LIN {X 0,Y 523.921,Z 257.848,A -85,B 0,C 180,E1 -4821.081,E2 -4821.081} C_VEL
LIN {X 0,Y 523.901,Z 257.849,A -85,B 0,C 180,E1 -4823.825,E2 -4823.825} C_VEL
LIN {X 0,Y 523.947,Z 257.848,A -85,B 0,C 180,E1 -4826.636,E2 -4826.636} C_VEL
LIN {X 0,Y 523.962,Z 257.841,A -85,B 0,C 180,E1 -4829.356,E2 -4829.356} C_VEL
LIN {X 0,Y 523.951,Z 257.849,A -85,B 0,C 180,E1 -4832.288,E2 -4832.288} C_VEL
LIN {X 0,Y 523.949,Z 257.848,A -85,B 0,C 180,E1 -4834.581,E2 -4834.581} C_VEL
LIN {X 0,Y 523.965,Z 257.93,A -85,B 0,C 180,E1 -4836.952,E2 -4836.952} C_VEL
LIN {X 0,Y 525.894,Z 266.836,A -85,B 0,C 180,E1 -4838.612,E2 -4838.612} C_VEL
LIN {X 0,Y 528.548,Z 277.959,A -85,B 0,C 180,E1 -4838.908,E2 -4838.908} C_VEL
LIN {X 0,Y 527.339,Z 416.797,A -85,B 0,C 180,E1 -4840.955,E2 -4840.955} C_VEL
LIN {X 0,Y 527.174,Z 435.165,A -85,B 0,C 180,E1 -4841.271,E2 -4841.271} C_VEL
LIN {X 0,Y 526.901,Z 450.096,A -85,B 0,C 180,E1 -4841.682,E2 -4841.682} C_VEL
LIN {X 0,Y 526.575,Z 464.31,A -85,B 0,C 180,E1 -4842.223,E2 -4842.223} C_VEL
LIN {X 0,Y 526.183,Z 478.273,A -85,B 0,C 180,E1 -4842.911,E2 -4842.911} C_VEL
LIN {X 0,Y 525.76,Z 492.557,A -85,B 0,C 180,E1 -4843.797,E2 -4843.797} C_VEL
LIN {X 0,Y 525.311,Z 505.414,A -85,B 0,C 180,E1 -4844.778,E2 -4844.778} C_VEL
LIN {X 0,Y 524.873,Z 517.153,A -85,B 0,C 180,E1 -4845.855,E2 -4845.855} C_VEL
LIN {X 0,Y 524.507,Z 527.829,A -85,B 0,C 180,E1 -4847.03,E2 -4847.03} C_VEL
LIN {X 0,Y 524.096,Z 538.235,A -85,B 0,C 180,E1 -4848.395,E2 -4848.395} C_VEL
LIN {X 0,Y 523.9,Z 546.784,A -85,B 0,C 180,E1 -4849.761,E2 -4849.761} C_VEL
LIN {X 0,Y 523.65,Z 553.936,A -85,B 0,C 180,E1 -4851.121,E2 -4851.121} C_VEL
LIN {X 0,Y 523.526,Z 560.464,A -85,B 0,C 180,E1 -4852.673,E2 -4852.673} C_VEL
LIN {X 0,Y 523.483,Z 565.622,A -85,B 0,C 180,E1 -4854.22,E2 -4854.22} C_VEL
LIN {X 0,Y 523.335,Z 568.597,A -85,B 0,C 180,E1 -4855.378,E2 -4855.378} C_VEL
LIN {X 0,Y 523.389,Z 571.449,A -85,B 0,C 180,E1 -4856.921,E2 -4856.921} C_VEL
LIN {X 0,Y 523.273,Z 573.167,A -85,B 0,C 180,E1 -4858.46,E2 -4858.46} C_VEL
LIN {X 0,Y 523.246,Z 573.806,A -85,B 0,C 180,E1 -4859.999,E2 -4859.999} C_VEL
LIN {X 0,Y 523.273,Z 573.231,A -85,B 0,C 180,E1 -4861.539,E2 -4861.539} C_VEL
LIN {X 0,Y 523.391,Z 571.557,A -85,B 0,C 180,E1 -4863.078,E2 -4863.078} C_VEL
LIN {X 0,Y 523.333,Z 568.774,A -85,B 0,C 180,E1 -4864.621,E2 -4864.621} C_VEL
LIN {X 0,Y 523.441,Z 564.656,A -85,B 0,C 180,E1 -4866.165,E2 -4866.165} C_VEL
LIN {X 0,Y 523.557,Z 559.289,A -85,B 0,C 180,E1 -4867.714,E2 -4867.714} C_VEL
LIN {X 0,Y 523.705,Z 552.375,A -85,B 0,C 180,E1 -4869.266,E2 -4869.266} C_VEL
LIN {X 0,Y 523.949,Z 544.953,A -85,B 0,C 180,E1 -4870.628,E2 -4870.628} C_VEL
LIN {X 0,Y 524.199,Z 536.232,A -85,B 0,C 180,E1 -4871.966,E2 -4871.966} C_VEL
LIN {X 0,Y 524.52,Z 526.84,A -85,B 0,C 180,E1 -4873.166,E2 -4873.166} C_VEL
LIN {X 0,Y 524.9,Z 516.03,A -85,B 0,C 180,E1 -4874.341,E2 -4874.341} C_VEL
LIN {X 0,Y 525.356,Z 503.897,A -85,B 0,C 180,E1 -4875.437,E2 -4875.437} C_VEL
LIN {X 0,Y 525.813,Z 491.098,A -85,B 0,C 180,E1 -4876.4,E2 -4876.4} C_VEL
LIN {X 0,Y 526.27,Z 478.382,A -85,B 0,C 180,E1 -4877.185,E2 -4877.185} C_VEL
LIN {X 0,Y 526.614,Z 464.639,A -85,B 0,C 180,E1 -4877.875,E2 -4877.875} C_VEL
LIN {X 0,Y 526.981,Z 448.493,A -85,B 0,C 180,E1 -4878.49,E2 -4878.49} C_VEL
LIN {X 0,Y 527.289,Z 433.513,A -85,B 0,C 180,E1 -4878.893,E2 -4878.893} C_VEL
LIN {X 0,Y 527.459,Z 412.098,A -85,B 0,C 180,E1 -4879.248,E2 -4879.248} C_VEL
LIN {X 0,Y 528.568,Z 278.087,A -85,B 0,C 180,E1 -4881.184,E2 -4881.184} C_VEL
LIN {X 0,Y 525.425,Z 265.012,A -85,B 0,C 180,E1 -4881.534,E2 -4881.534} C_VEL
LIN {X 0,Y 523.937,Z 257.848,A -85,B 0,C 180,E1 -4882.812,E2 -4882.812} C_VEL
LIN {X 0,Y 523.91,Z 257.851,A -85,B 0,C 180,E1 -4883.324,E2 -4883.324} C_VEL
LIN {X 0,Y 523.244,Z 257.937,A -85,B 0,C 180,E1 -4883.965,E2 -4883.965} C_VEL
LIN {X 0,Y 520.418,Z 258.288,A -85,B 0,C 180,E1 -4885.006,E2 -4885.006} C_VEL
LIN {X 0,Y 518.024,Z 258.585,A -85,B 0,C 180,E1 -4885.845,E2 -4885.845} C_VEL
LIN {X 0,Y 516.984,Z 258.71,A -85,B 0,C 180,E1 -4886.492,E2 -4886.492} C_VEL
LIN {X 0,Y 516.893,Z 258.72,A -85,B 0,C 180,E1 -4886.711,E2 -4886.711} C_VEL
LIN {X 0,Y 516.909,Z 258.721,A -85,B 0,C 180,E1 -4889.522,E2 -4889.522} C_VEL
LIN {X 0,Y 516.895,Z 258.719,A -85,B 0,C 180,E1 -4892.542,E2 -4892.542} C_VEL
LIN {X 0,Y 516.863,Z 258.724,A -85,B 0,C 180,E1 -4895.328,E2 -4895.328} C_VEL
LIN {X 0,Y 516.877,Z 258.728,A -85,B 0,C 180,E1 -4897.942,E2 -4897.942} C_VEL
LIN {X 0,Y 516.881,Z 258.72,A -85,B 0,C 180,E1 -4900.741,E2 -4900.741} C_VEL
LIN {X 0,Y 516.861,Z 258.722,A -85,B 0,C 180,E1 -4902.832,E2 -4902.832} C_VEL
LIN {X 0,Y 516.893,Z 258.718,A -85,B 0,C 180,E1 -4905.006,E2 -4905.006} C_VEL
LIN {X 0,Y 516.911,Z 258.718,A -85,B 0,C 180,E1 -4908.398,E2 -4908.398} C_VEL
LIN {X 0,Y 516.877,Z 258.723,A -85,B 0,C 180,E1 -4911.283,E2 -4911.283} C_VEL
LIN {X 0,Y 516.868,Z 258.724,A -85,B 0,C 180,E1 -4914.219,E2 -4914.219} C_VEL
LIN {X 0,Y 516.877,Z 258.721,A -85,B 0,C 180,E1 -4917.051,E2 -4917.051} C_VEL
LIN {X 0,Y 516.887,Z 258.727,A -85,B 0,C 180,E1 -4919.795,E2 -4919.795} C_VEL
LIN {X 0,Y 516.895,Z 258.719,A -85,B 0,C 180,E1 -4922.465,E2 -4922.465} C_VEL
LIN {X 0,Y 516.861,Z 258.723,A -85,B 0,C 180,E1 -4925.068,E2 -4925.068} C_VEL
LIN {X 0,Y 516.863,Z 258.73,A -85,B 0,C 180,E1 -4927.62,E2 -4927.62} C_VEL
LIN {X 0,Y 516.925,Z 258.717,A -85,B 0,C 180,E1 -4930.129,E2 -4930.129} C_VEL
LIN {X 0,Y 516.901,Z 258.717,A -85,B 0,C 180,E1 -4932.594,E2 -4932.594} C_VEL
LIN {X 0,Y 516.935,Z 258.714,A -85,B 0,C 180,E1 -4935.029,E2 -4935.029} C_VEL
LIN {X 0,Y 516.959,Z 258.711,A -85,B 0,C 180,E1 -4938.233,E2 -4938.233} C_VEL
LIN {X 0,Y 516.961,Z 258.716,A -85,B 0,C 180,E1 -4941.399,E2 -4941.399} C_VEL
LIN {X 0,Y 516.993,Z 258.712,A -85,B 0,C 180,E1 -4943.756,E2 -4943.756} C_VEL
LIN {X 0,Y 517.003,Z 258.705,A -85,B 0,C 180,E1 -4946.882,E2 -4946.882} C_VEL
LIN {X 0,Y 517.072,Z 258.699,A -85,B 0,C 180,E1 -4949.999,E2 -4949.999} C_VEL
LIN {X 0,Y 517.004,Z 258.708,A -85,B 0,C 180,E1 -4953.116,E2 -4953.116} C_VEL
LIN {X 0,Y 516.992,Z 258.707,A -85,B 0,C 180,E1 -4956.242,E2 -4956.242} C_VEL
LIN {X 0,Y 516.938,Z 258.72,A -85,B 0,C 180,E1 -4959.388,E2 -4959.388} C_VEL
LIN {X 0,Y 516.941,Z 258.717,A -85,B 0,C 180,E1 -4961.806,E2 -4961.806} C_VEL
LIN {X 0,Y 516.933,Z 258.718,A -85,B 0,C 180,E1 -4965.145,E2 -4965.145} C_VEL
LIN {X 0,Y 516.913,Z 258.716,A -85,B 0,C 180,E1 -4968.221,E2 -4968.221} C_VEL
LIN {X 0,Y 516.9,Z 258.718,A -85,B 0,C 180,E1 -4970.701,E2 -4970.701} C_VEL
LIN {X 0,Y 516.878,Z 258.721,A -85,B 0,C 180,E1 -4974.072,E2 -4974.072} C_VEL
LIN {X 0,Y 516.913,Z 258.716,A -85,B 0,C 180,E1 -4976.657,E2 -4976.657} C_VEL
LIN {X 0,Y 516.897,Z 258.725,A -85,B 0,C 180,E1 -4979.523,E2 -4979.523} C_VEL
LIN {X 0,Y 516.887,Z 258.719,A -85,B 0,C 180,E1 -4982.544,E2 -4982.544} C_VEL
LIN {X 0,Y 516.867,Z 258.731,A -85,B 0,C 180,E1 -4985.331,E2 -4985.331} C_VEL
LIN {X 0,Y 516.867,Z 258.723,A -85,B 0,C 180,E1 -4987.943,E2 -4987.943} C_VEL
LIN {X 0,Y 516.87,Z 258.723,A -85,B 0,C 180,E1 -4990.741,E2 -4990.741} C_VEL
LIN {X 0,Y 516.889,Z 258.721,A -85,B 0,C 180,E1 -4992.829,E2 -4992.829} C_VEL
LIN {X 0,Y 516.908,Z 258.721,A -85,B 0,C 180,E1 -4995.01,E2 -4995.01} C_VEL
LIN {X 0,Y 516.9,Z 258.717,A -85,B 0,C 180,E1 -4998.398,E2 -4998.398} C_VEL
LIN {X 0,Y 516.867,Z 258.73,A -85,B 0,C 180,E1 -5001.284,E2 -5001.284} C_VEL
LIN {X 0,Y 516.873,Z 258.721,A -85,B 0,C 180,E1 -5004.221,E2 -5004.221} C_VEL
LIN {X 0,Y 516.882,Z 258.726,A -85,B 0,C 180,E1 -5007.053,E2 -5007.053} C_VEL
LIN {X 0,Y 516.877,Z 258.722,A -85,B 0,C 180,E1 -5009.796,E2 -5009.796} C_VEL
LIN {X 0,Y 516.912,Z 258.717,A -85,B 0,C 180,E1 -5012.467,E2 -5012.467} C_VEL
LIN {X 0,Y 516.893,Z 258.726,A -85,B 0,C 180,E1 -5015.072,E2 -5015.072} C_VEL
LIN {X 0,Y 516.872,Z 258.722,A -85,B 0,C 180,E1 -5018.463,E2 -5018.463} C_VEL
LIN {X 0,Y 516.888,Z 258.725,A -85,B 0,C 180,E1 -5020.955,E2 -5020.955} C_VEL
LIN {X 0,Y 516.899,Z 258.722,A -85,B 0,C 180,E1 -5023.411,E2 -5023.411} C_VEL
LIN {X 0,Y 516.879,Z 258.721,A -85,B 0,C 180,E1 -5025.834,E2 -5025.834} C_VEL
LIN {X 0,Y 516.951,Z 258.711,A -85,B 0,C 180,E1 -5028.234,E2 -5028.234} C_VEL
LIN {X 0,Y 516.951,Z 258.715,A -85,B 0,C 180,E1 -5031.4,E2 -5031.4} C_VEL
LIN {X 0,Y 516.988,Z 258.707,A -85,B 0,C 180,E1 -5033.757,E2 -5033.757} C_VEL
LIN {X 0,Y 517.001,Z 258.712,A -85,B 0,C 180,E1 -5036.884,E2 -5036.884} C_VEL
LIN {X 0,Y 517.067,Z 258.696,A -85,B 0,C 180,E1 -5040.001,E2 -5040.001} C_VEL
LIN {X 0,Y 517.001,Z 258.712,A -85,B 0,C 180,E1 -5043.118,E2 -5043.118} C_VEL
LIN {X 0,Y 516.987,Z 258.707,A -85,B 0,C 180,E1 -5046.244,E2 -5046.244} C_VEL
LIN {X 0,Y 516.941,Z 258.715,A -85,B 0,C 180,E1 -5049.39,E2 -5049.39} C_VEL
LIN {X 0,Y 516.942,Z 258.712,A -85,B 0,C 180,E1 -5051.809,E2 -5051.809} C_VEL
LIN {X 0,Y 516.932,Z 258.719,A -85,B 0,C 180,E1 -5055.147,E2 -5055.147} C_VEL
LIN {X 0,Y 516.913,Z 258.717,A -85,B 0,C 180,E1 -5058.223,E2 -5058.223} C_VEL
LIN {X 0,Y 516.902,Z 258.723,A -85,B 0,C 180,E1 -5060.702,E2 -5060.702} C_VEL
LIN {X 0,Y 516.892,Z 258.719,A -85,B 0,C 180,E1 -5064.073,E2 -5064.073} C_VEL
LIN {X 0,Y 516.913,Z 258.722,A -85,B 0,C 180,E1 -5066.659,E2 -5066.659} C_VEL
LIN {X 0,Y 516.901,Z 258.718,A -85,B 0,C 180,E1 -5069.525,E2 -5069.525} C_VEL
LIN {X 0,Y 516.885,Z 258.724,A -85,B 0,C 180,E1 -5072.544,E2 -5072.544} C_VEL
LIN {X 0,Y 516.859,Z 258.725,A -85,B 0,C 180,E1 -5075.331,E2 -5075.331} C_VEL
LIN {X 0,Y 516.871,Z 258.721,A -85,B 0,C 180,E1 -5077.944,E2 -5077.944} C_VEL
LIN {X 0,Y 516.875,Z 258.729,A -85,B 0,C 180,E1 -5080.743,E2 -5080.743} C_VEL
LIN {X 0,Y 516.875,Z 258.729,A -85,B 0,C 180,E1 -5082.833,E2 -5082.833} C_VEL
LIN {X 0,Y 516.887,Z 258.724,A -85,B 0,C 180,E1 -5085.008,E2 -5085.008} C_VEL
LIN {X 0,Y 516.906,Z 258.721,A -85,B 0,C 180,E1 -5088.4,E2 -5088.4} C_VEL
LIN {X 0,Y 516.874,Z 258.723,A -85,B 0,C 180,E1 -5091.285,E2 -5091.285} C_VEL
LIN {X 0,Y 516.861,Z 258.725,A -85,B 0,C 180,E1 -5094.221,E2 -5094.221} C_VEL
LIN {X 0,Y 516.889,Z 258.723,A -85,B 0,C 180,E1 -5097.054,E2 -5097.054} C_VEL
LIN {X 0,Y 516.908,Z 258.724,A -85,B 0,C 180,E1 -5100.275,E2 -5100.275} C_VEL
LIN {X 0,Y 520.469,Z 273.636,A -85,B 0,C 180,E1 -5102.454,E2 -5102.454} C_VEL
LIN {X 0,Y 519.948,Z 291.889,A -85,B 0,C 180,E1 -5104.753,E2 -5104.753} C_VEL
LIN {X 0,Y 519.149,Z 315.846,A -85,B 0,C 180,E1 -5107.726,E2 -5107.726} C_VEL
LIN {X 0,Y 519.053,Z 320.097,A -85,B 0,C 180,E1 -5108.227,E2 -5108.227} C_VEL
LIN {X 0,Y 521.792,Z 336.231,A -85,B 0,C 180,E1 -5108.604,E2 -5108.604} C_VEL
LIN {X 0,Y 521.279,Z 401.8,A -85,B 0,C 180,E1 -5109.558,E2 -5109.558} C_VEL
LIN {X 0,Y 520.628,Z 477.491,A -85,B 0,C 180,E1 -5110.663,E2 -5110.663} C_VEL
LIN {X 0,Y 520.418,Z 493.511,A -85,B 0,C 180,E1 -5110.965,E2 -5110.965} C_VEL
LIN {X 0,Y 520.015,Z 508.842,A -85,B 0,C 180,E1 -5111.411,E2 -5111.411} C_VEL
LIN {X 0,Y 519.549,Z 524.172,A -85,B 0,C 180,E1 -5112.027,E2 -5112.027} C_VEL
LIN {X 0,Y 519.139,Z 538.471,A -85,B 0,C 180,E1 -5112.775,E2 -5112.775} C_VEL
LIN {X 0,Y 518.598,Z 552.246,A -85,B 0,C 180,E1 -5113.669,E2 -5113.669} C_VEL
LIN {X 0,Y 518.144,Z 565.469,A -85,B 0,C 180,E1 -5114.718,E2 -5114.718} C_VEL
LIN {X 0,Y 517.634,Z 577.41,A -85,B 0,C 180,E1 -5115.856,E2 -5115.856} C_VEL
LIN {X 0,Y 517.3,Z 587.893,A -85,B 0,C 180,E1 -5117.047,E2 -5117.047} C_VEL
LIN {X 0,Y 516.926,Z 597.578,A -85,B 0,C 180,E1 -5118.351,E2 -5118.351} C_VEL
LIN {X 0,Y 516.772,Z 605.519,A -85,B 0,C 180,E1 -5119.62,E2 -5119.62} C_VEL
LIN {X 0,Y 516.546,Z 612.786,A -85,B 0,C 180,E1 -5120.999,E2 -5120.999} C_VEL
LIN {X 0,Y 516.391,Z 619.514,A -85,B 0,C 180,E1 -5122.572,E2 -5122.572} C_VEL
LIN {X 0,Y 516.374,Z 624.776,A -85,B 0,C 180,E1 -5124.142,E2 -5124.142} C_VEL
LIN {X 0,Y 516.238,Z 627.805,A -85,B 0,C 180,E1 -5125.316,E2 -5125.316} C_VEL
LIN {X 0,Y 516.272,Z 630.767,A -85,B 0,C 180,E1 -5126.88,E2 -5126.88} C_VEL
LIN {X 0,Y 516.189,Z 632.523,A -85,B 0,C 180,E1 -5128.441,E2 -5128.441} C_VEL
LIN {X 0,Y 516.154,Z 633.12,A -85,B 0,C 180,E1 -5130.001,E2 -5130.001} C_VEL
LIN {X 0,Y 516.189,Z 632.512,A -85,B 0,C 180,E1 -5131.561,E2 -5131.561} C_VEL
LIN {X 0,Y 516.272,Z 630.738,A -85,B 0,C 180,E1 -5133.122,E2 -5133.122} C_VEL
LIN {X 0,Y 516.239,Z 627.76,A -85,B 0,C 180,E1 -5134.686,E2 -5134.686} C_VEL
LIN {X 0,Y 516.373,Z 624.721,A -85,B 0,C 180,E1 -5135.86,E2 -5135.86} C_VEL
LIN {X 0,Y 516.41,Z 619.425,A -85,B 0,C 180,E1 -5137.429,E2 -5137.429} C_VEL
LIN {X 0,Y 516.547,Z 612.637,A -85,B 0,C 180,E1 -5139.003,E2 -5139.003} C_VEL
LIN {X 0,Y 516.774,Z 605.303,A -85,B 0,C 180,E1 -5140.382,E2 -5140.382} C_VEL
LIN {X 0,Y 516.988,Z 596.054,A -85,B 0,C 180,E1 -5141.825,E2 -5141.825} C_VEL
LIN {X 0,Y 517.332,Z 585.798,A -85,B 0,C 180,E1 -5143.154,E2 -5143.154} C_VEL
LIN {X 0,Y 517.749,Z 573.832,A -85,B 0,C 180,E1 -5144.444,E2 -5144.444} C_VEL
LIN {X 0,Y 518.169,Z 561.862,A -85,B 0,C 180,E1 -5145.521,E2 -5145.521} C_VEL
LIN {X 0,Y 518.609,Z 548.271,A -85,B 0,C 180,E1 -5146.535,E2 -5146.535} C_VEL
LIN {X 0,Y 519.133,Z 535.278,A -85,B 0,C 180,E1 -5147.329,E2 -5147.329} C_VEL
LIN {X 0,Y 519.518,Z 521.199,A -85,B 0,C 180,E1 -5148.027,E2 -5148.027} C_VEL
LIN {X 0,Y 519.915,Z 505.833,A -85,B 0,C 180,E1 -5148.613,E2 -5148.613} C_VEL
LIN {X 0,Y 520.244,Z 490.363,A -85,B 0,C 180,E1 -5149.034,E2 -5149.034} C_VEL
LIN {X 0,Y 520.483,Z 468.714,A -85,B 0,C 180,E1 -5149.396,E2 -5149.396} C_VEL
LIN {X 0,Y 521.504,Z 356.758,A -85,B 0,C 180,E1 -5151.055,E2 -5151.055} C_VEL
LIN {X 0,Y 521.615,Z 334.909,A -85,B 0,C 180,E1 -5151.398,E2 -5151.398} C_VEL
LIN {X 0,Y 518.743,Z 318.086,A -85,B 0,C 180,E1 -5151.804,E2 -5151.804} C_VEL
LIN {X 0,Y 519.346,Z 297.016,A -85,B 0,C 180,E1 -5154.378,E2 -5154.378} C_VEL
LIN {X 0,Y 520.048,Z 275.766,A -85,B 0,C 180,E1 -5157.039,E2 -5157.039} C_VEL
LIN {X 0,Y 519.935,Z 271.638,A -85,B 0,C 180,E1 -5157.579,E2 -5157.579} C_VEL
LIN {X 0,Y 516.911,Z 258.725,A -85,B 0,C 180,E1 -5159.491,E2 -5159.491} C_VEL
LIN {X 0,Y 516.9,Z 258.725,A -85,B 0,C 180,E1 -5162.544,E2 -5162.544} C_VEL
LIN {X 0,Y 516.871,Z 258.73,A -85,B 0,C 180,E1 -5165.33,E2 -5165.33} C_VEL
LIN {X 0,Y 516.886,Z 258.723,A -85,B 0,C 180,E1 -5167.943,E2 -5167.943} C_VEL
LIN {X 0,Y 516.888,Z 258.727,A -85,B 0,C 180,E1 -5170.742,E2 -5170.742} C_VEL
LIN {X 0,Y 516.888,Z 258.728,A -85,B 0,C 180,E1 -5172.832,E2 -5172.832} C_VEL
LIN {X 0,Y 516.929,Z 258.722,A -85,B 0,C 180,E1 -5175.01,E2 -5175.01} C_VEL
LIN {X 0,Y 516.919,Z 258.722,A -85,B 0,C 180,E1 -5178.399,E2 -5178.399} C_VEL
LIN {X 0,Y 516.885,Z 258.723,A -85,B 0,C 180,E1 -5181.284,E2 -5181.284} C_VEL
LIN {X 0,Y 516.873,Z 258.728,A -85,B 0,C 180,E1 -5184.219,E2 -5184.219} C_VEL
LIN {X 0,Y 516.901,Z 258.722,A -85,B 0,C 180,E1 -5187.053,E2 -5187.053} C_VEL
LIN {X 0,Y 516.897,Z 258.723,A -85,B 0,C 180,E1 -5189.796,E2 -5189.796} C_VEL
LIN {X 0,Y 516.904,Z 258.726,A -85,B 0,C 180,E1 -5192.466,E2 -5192.466} C_VEL
LIN {X 0,Y 516.878,Z 258.727,A -85,B 0,C 180,E1 -5195.07,E2 -5195.07} C_VEL
LIN {X 0,Y 516.901,Z 258.826,A -85,B 0,C 180,E1 -5196.645,E2 -5196.645} C_VEL
LIN {X 0,Y 518.909,Z 267.547,A -85,B 0,C 180,E1 -5198.312,E2 -5198.312} C_VEL
LIN {X 0,Y 521.248,Z 276.054,A -85,B 0,C 180,E1 -5198.56,E2 -5198.56} C_VEL
LIN {X 0,Y 521.956,Z 279.772,A -85,B 0,C 180,E1 -5198.653,E2 -5198.653} C_VEL
LIN {X 0,Y 520.595,Z 407.846,A -85,B 0,C 180,E1 -5200.6,E2 -5200.6} C_VEL
LIN {X 0,Y 520.376,Z 432.757,A -85,B 0,C 180,E1 -5200.994,E2 -5200.994} C_VEL
LIN {X 0,Y 520.151,Z 448.088,A -85,B 0,C 180,E1 -5201.395,E2 -5201.395} C_VEL
LIN {X 0,Y 519.803,Z 462.708,A -85,B 0,C 180,E1 -5201.933,E2 -5201.933} C_VEL
LIN {X 0,Y 519.413,Z 476.248,A -85,B 0,C 180,E1 -5202.58,E2 -5202.58} C_VEL
LIN {X 0,Y 519.026,Z 489.585,A -85,B 0,C 180,E1 -5203.378,E2 -5203.378} C_VEL
LIN {X 0,Y 518.536,Z 501.867,A -85,B 0,C 180,E1 -5204.272,E2 -5204.272} C_VEL
LIN {X 0,Y 518.083,Z 514.292,A -85,B 0,C 180,E1 -5205.365,E2 -5205.365} C_VEL
LIN {X 0,Y 517.707,Z 524.664,A -85,B 0,C 180,E1 -5206.457,E2 -5206.457} C_VEL
LIN {X 0,Y 517.279,Z 534.383,A -85,B 0,C 180,E1 -5207.663,E2 -5207.663} C_VEL
LIN {X 0,Y 517.026,Z 543.598,A -85,B 0,C 180,E1 -5209.029,E2 -5209.029} C_VEL
LIN {X 0,Y 516.74,Z 550.337,A -85,B 0,C 180,E1 -5210.211,E2 -5210.211} C_VEL
LIN {X 0,Y 516.557,Z 557.748,A -85,B 0,C 180,E1 -5211.786,E2 -5211.786} C_VEL
LIN {X 0,Y 516.428,Z 563.866,A -85,B 0,C 180,E1 -5213.441,E2 -5213.441} C_VEL
LIN {X 0,Y 516.378,Z 567.075,A -85,B 0,C 180,E1 -5214.533,E2 -5214.533} C_VEL
LIN {X 0,Y 516.328,Z 570.555,A -85,B 0,C 180,E1 -5216.097,E2 -5216.097} C_VEL
LIN {X 0,Y 516.259,Z 572.897,A -85,B 0,C 180,E1 -5217.659,E2 -5217.659} C_VEL
LIN {X 0,Y 516.162,Z 574.03,A -85,B 0,C 180,E1 -5219.219,E2 -5219.219} C_VEL
LIN {X 0,Y 516.163,Z 574.041,A -85,B 0,C 180,E1 -5220.78,E2 -5220.78} C_VEL
LIN {X 0,Y 516.261,Z 572.958,A -85,B 0,C 180,E1 -5222.34,E2 -5222.34} C_VEL
LIN {X 0,Y 516.328,Z 570.666,A -85,B 0,C 180,E1 -5223.902,E2 -5223.902} C_VEL
LIN {X 0,Y 516.374,Z 567.226,A -85,B 0,C 180,E1 -5225.466,E2 -5225.466} C_VEL
LIN {X 0,Y 516.431,Z 562.48,A -85,B 0,C 180,E1 -5227.035,E2 -5227.035} C_VEL
LIN {X 0,Y 516.57,Z 556.314,A -85,B 0,C 180,E1 -5228.606,E2 -5228.606} C_VEL
LIN {X 0,Y 516.771,Z 548.572,A -85,B 0,C 180,E1 -5230.183,E2 -5230.183} C_VEL
LIN {X 0,Y 517.047,Z 540.255,A -85,B 0,C 180,E1 -5231.565,E2 -5231.565} C_VEL
LIN {X 0,Y 517.431,Z 530.257,A -85,B 0,C 180,E1 -5232.95,E2 -5232.95} C_VEL
LIN {X 0,Y 517.848,Z 519.954,A -85,B 0,C 180,E1 -5234.139,E2 -5234.139} C_VEL
LIN {X 0,Y 518.32,Z 508.122,A -85,B 0,C 180,E1 -5235.29,E2 -5235.29} C_VEL
LIN {X 0,Y 518.793,Z 495.53,A -85,B 0,C 180,E1 -5236.305,E2 -5236.305} C_VEL
LIN {X 0,Y 519.327,Z 481.733,A -85,B 0,C 180,E1 -5237.219,E2 -5237.219} C_VEL
LIN {X 0,Y 519.734,Z 467.644,A -85,B 0,C 180,E1 -5237.967,E2 -5237.967} C_VEL
LIN {X 0,Y 520.142,Z 452.164,A -85,B 0,C 180,E1 -5238.601,E2 -5238.601} C_VEL
LIN {X 0,Y 520.457,Z 436.707,A -85,B 0,C 180,E1 -5239.057,E2 -5239.057} C_VEL
LIN {X 0,Y 520.664,Z 420.56,A -85,B 0,C 180,E1 -5239.362,E2 -5239.362} C_VEL
LIN {X 0,Y 521.941,Z 279.769,A -85,B 0,C 180,E1 -5241.441,E2 -5241.441} C_VEL
LIN {X 0,Y 519.648,Z 269.401,A -85,B 0,C 180,E1 -5241.704,E2 -5241.704} C_VEL
LIN {X 0,Y 518.278,Z 265.35,A -85,B 0,C 180,E1 -5241.837,E2 -5241.837} C_VEL
LIN {X 0,Y 516.887,Z 258.727,A -85,B 0,C 180,E1 -5243.021,E2 -5243.021} C_VEL
LIN {X 0,Y 516.899,Z 258.724,A -85,B 0,C 180,E1 -5246.185,E2 -5246.185} C_VEL
LIN {X 0,Y 516.893,Z 258.72,A -85,B 0,C 180,E1 -5246.711,E2 -5246.711} C_VEL
LIN {X 0,Y 516.209,Z 258.807,A -85,B 0,C 180,E1 -5247.362,E2 -5247.362} C_VEL
LIN {X 0,Y 513.356,Z 259.163,A -85,B 0,C 180,E1 -5248.418,E2 -5248.418} C_VEL
LIN {X 0,Y 510.954,Z 259.464,A -85,B 0,C 180,E1 -5249.269,E2 -5249.269} C_VEL
LIN {X 0,Y 509.92,Z 259.595,A -85,B 0,C 180,E1 -5249.926,E2 -5249.926} C_VEL
LIN {X 0,Y 509.835,Z 259.601,A -85,B 0,C 180,E1 -5250.148,E2 -5250.148} C_VEL
LIN {X 0,Y 509.858,Z 259.598,A -85,B 0,C 180,E1 -5253.46,E2 -5253.46} C_VEL
LIN {X 0,Y 509.808,Z 259.603,A -85,B 0,C 180,E1 -5256.353,E2 -5256.353} C_VEL
LIN {X 0,Y 509.844,Z 259.599,A -85,B 0,C 180,E1 -5259.351,E2 -5259.351} C_VEL
LIN {X 0,Y 509.818,Z 259.601,A -85,B 0,C 180,E1 -5262.49,E2 -5262.49} C_VEL
LIN {X 0,Y 509.837,Z 259.6,A -85,B 0,C 180,E1 -5265.329,E2 -5265.329} C_VEL
LIN {X 0,Y 509.853,Z 259.596,A -85,B 0,C 180,E1 -5268.573,E2 -5268.573} C_VEL
LIN {X 0,Y 509.847,Z 259.605,A -85,B 0,C 180,E1 -5271.785,E2 -5271.785} C_VEL
LIN {X 0,Y 509.826,Z 259.599,A -85,B 0,C 180,E1 -5274.621,E2 -5274.621} C_VEL
LIN {X 0,Y 509.856,Z 259.6,A -85,B 0,C 180,E1 -5277.48,E2 -5277.48} C_VEL
LIN {X 0,Y 509.854,Z 259.597,A -85,B 0,C 180,E1 -5280.273,E2 -5280.273} C_VEL
LIN {X 0,Y 509.879,Z 259.6,A -85,B 0,C 180,E1 -5283.627,E2 -5283.627} C_VEL
LIN {X 0,Y 509.816,Z 259.6,A -85,B 0,C 180,E1 -5286.435,E2 -5286.435} C_VEL
LIN {X 0,Y 509.911,Z 259.595,A -85,B 0,C 180,E1 -5289.844,E2 -5289.844} C_VEL
LIN {X 0,Y 509.869,Z 259.596,A -85,B 0,C 180,E1 -5293.173,E2 -5293.173} C_VEL
LIN {X 0,Y 509.856,Z 259.604,A -85,B 0,C 180,E1 -5295.633,E2 -5295.633} C_VEL
LIN {X 0,Y 509.905,Z 259.589,A -85,B 0,C 180,E1 -5298.873,E2 -5298.873} C_VEL
LIN {X 0,Y 509.944,Z 259.586,A -85,B 0,C 180,E1 -5302.077,E2 -5302.077} C_VEL
LIN {X 0,Y 509.97,Z 259.581,A -85,B 0,C 180,E1 -5304.463,E2 -5304.463} C_VEL
LIN {X 0,Y 510.044,Z 259.58,A -85,B 0,C 180,E1 -5307.63,E2 -5307.63} C_VEL
LIN {X 0,Y 510.043,Z 259.574,A -85,B 0,C 180,E1 -5309.999,E2 -5309.999} C_VEL
LIN {X 0,Y 510.042,Z 259.572,A -85,B 0,C 180,E1 -5312.368,E2 -5312.368} C_VEL
LIN {X 0,Y 509.968,Z 259.59,A -85,B 0,C 180,E1 -5315.535,E2 -5315.535} C_VEL
LIN {X 0,Y 509.94,Z 259.588,A -85,B 0,C 180,E1 -5317.921,E2 -5317.921} C_VEL
LIN {X 0,Y 509.902,Z 259.593,A -85,B 0,C 180,E1 -5321.124,E2 -5321.124} C_VEL
LIN {X 0,Y 509.852,Z 259.595,A -85,B 0,C 180,E1 -5324.365,E2 -5324.365} C_VEL
LIN {X 0,Y 509.882,Z 259.598,A -85,B 0,C 180,E1 -5327.651,E2 -5327.651} C_VEL
LIN {X 0,Y 509.874,Z 259.593,A -85,B 0,C 180,E1 -5330.401,E2 -5330.401} C_VEL
LIN {X 0,Y 509.81,Z 259.607,A -85,B 0,C 180,E1 -5333.563,E2 -5333.563} C_VEL
LIN {X 0,Y 509.898,Z 259.59,A -85,B 0,C 180,E1 -5336.378,E2 -5336.378} C_VEL
LIN {X 0,Y 509.863,Z 259.596,A -85,B 0,C 180,E1 -5338.844,E2 -5338.844} C_VEL
LIN {X 0,Y 509.812,Z 259.606,A -85,B 0,C 180,E1 -5341.589,E2 -5341.589} C_VEL
LIN {X 0,Y 509.839,Z 259.597,A -85,B 0,C 180,E1 -5344.413,E2 -5344.413} C_VEL
LIN {X 0,Y 509.804,Z 259.611,A -85,B 0,C 180,E1 -5347.34,E2 -5347.34} C_VEL
LIN {X 0,Y 509.823,Z 259.599,A -85,B 0,C 180,E1 -5350.382,E2 -5350.382} C_VEL
LIN {X 0,Y 509.825,Z 259.604,A -85,B 0,C 180,E1 -5353.064,E2 -5353.064} C_VEL
LIN {X 0,Y 509.816,Z 259.602,A -85,B 0,C 180,E1 -5355.792,E2 -5355.792} C_VEL
LIN {X 0,Y 509.841,Z 259.598,A -85,B 0,C 180,E1 -5358.574,E2 -5358.574} C_VEL
LIN {X 0,Y 509.836,Z 259.599,A -85,B 0,C 180,E1 -5361.786,E2 -5361.786} C_VEL
LIN {X 0,Y 509.828,Z 259.6,A -85,B 0,C 180,E1 -5364.623,E2 -5364.623} C_VEL
LIN {X 0,Y 509.851,Z 259.601,A -85,B 0,C 180,E1 -5367.481,E2 -5367.481} C_VEL
LIN {X 0,Y 509.843,Z 259.596,A -85,B 0,C 180,E1 -5370.274,E2 -5370.274} C_VEL
LIN {X 0,Y 509.87,Z 259.599,A -85,B 0,C 180,E1 -5372.944,E2 -5372.944} C_VEL
LIN {X 0,Y 509.849,Z 259.599,A -85,B 0,C 180,E1 -5375.574,E2 -5375.574} C_VEL
LIN {X 0,Y 509.836,Z 259.604,A -85,B 0,C 180,E1 -5378.999,E2 -5378.999} C_VEL
LIN {X 0,Y 509.874,Z 259.593,A -85,B 0,C 180,E1 -5381.999,E2 -5381.999} C_VEL
LIN {X 0,Y 509.896,Z 259.595,A -85,B 0,C 180,E1 -5384.819,E2 -5384.819} C_VEL
LIN {X 0,Y 509.886,Z 259.591,A -85,B 0,C 180,E1 -5388.125,E2 -5388.125} C_VEL
LIN {X 0,Y 509.897,Z 259.596,A -85,B 0,C 180,E1 -5391.28,E2 -5391.28} C_VEL
LIN {X 0,Y 509.94,Z 259.586,A -85,B 0,C 180,E1 -5393.671,E2 -5393.671} C_VEL
LIN {X 0,Y 509.943,Z 259.59,A -85,B 0,C 180,E1 -5396.84,E2 -5396.84} C_VEL
LIN {X 0,Y 510.052,Z 259.577,A -85,B 0,C 180,E1 -5399.211,E2 -5399.211} C_VEL
LIN {X 0,Y 509.917,Z 259.589,A -85,B 0,C 180,E1 -5401.58,E2 -5401.58} C_VEL
LIN {X 0,Y 509.942,Z 259.591,A -85,B 0,C 180,E1 -5403.161,E2 -5403.161} C_VEL
LIN {X 0,Y 509.939,Z 259.586,A -85,B 0,C 180,E1 -5406.331,E2 -5406.331} C_VEL
LIN {X 0,Y 509.904,Z 259.594,A -85,B 0,C 180,E1 -5408.721,E2 -5408.721} C_VEL
LIN {X 0,Y 509.892,Z 259.59,A -85,B 0,C 180,E1 -5411.932,E2 -5411.932} C_VEL
LIN {X 0,Y 509.882,Z 259.596,A -85,B 0,C 180,E1 -5415.243,E2 -5415.243} C_VEL
LIN {X 0,Y 509.87,Z 259.593,A -85,B 0,C 180,E1 -5417.999,E2 -5417.999} C_VEL
LIN {X 0,Y 509.84,Z 259.604,A -85,B 0,C 180,E1 -5421.003,E2 -5421.003} C_VEL
LIN {X 0,Y 509.851,Z 259.598,A -85,B 0,C 180,E1 -5424.427,E2 -5424.427} C_VEL
LIN {X 0,Y 509.872,Z 259.599,A -85,B 0,C 180,E1 -5427.057,E2 -5427.057} C_VEL
LIN {X 0,Y 509.847,Z 259.596,A -85,B 0,C 180,E1 -5429.752,E2 -5429.752} C_VEL
LIN {X 0,Y 509.863,Z 259.603,A -85,B 0,C 180,E1 -5432.775,E2 -5432.775} C_VEL
LIN {X 0,Y 509.818,Z 259.6,A -85,B 0,C 180,E1 -5435.58,E2 -5435.58} C_VEL
LIN {X 0,Y 509.84,Z 259.6,A -85,B 0,C 180,E1 -5438.339,E2 -5438.339} C_VEL
LIN {X 0,Y 509.848,Z 259.597,A -85,B 0,C 180,E1 -5441.427,E2 -5441.427} C_VEL
LIN {X 0,Y 509.831,Z 259.606,A -85,B 0,C 180,E1 -5444.671,E2 -5444.671} C_VEL
LIN {X 0,Y 509.825,Z 259.599,A -85,B 0,C 180,E1 -5447.511,E2 -5447.511} C_VEL
LIN {X 0,Y 509.84,Z 259.606,A -85,B 0,C 180,E1 -5450.649,E2 -5450.649} C_VEL
LIN {X 0,Y 509.803,Z 259.602,A -85,B 0,C 180,E1 -5453.647,E2 -5453.647} C_VEL
LIN {X 0,Y 509.853,Z 259.601,A -85,B 0,C 180,E1 -5456.54,E2 -5456.54} C_VEL
LIN {X 0,Y 509.858,Z 259.601,A -85,B 0,C 180,E1 -5459.966,E2 -5459.966} C_VEL
LIN {X 0,Y 509.876,Z 259.68,A -85,B 0,C 180,E1 -5460.025,E2 -5460.025} C_VEL
LIN {X 0,Y 513.607,Z 275.06,A -85,B 0,C 180,E1 -5462.276,E2 -5462.276} C_VEL
LIN {X 0,Y 513.51,Z 281.809,A -85,B 0,C 180,E1 -5463.152,E2 -5463.152} C_VEL
LIN {X 0,Y 512.657,Z 305.432,A -85,B 0,C 180,E1 -5466.147,E2 -5466.147} C_VEL
LIN {X 0,Y 512.142,Z 319.536,A -85,B 0,C 180,E1 -5467.911,E2 -5467.911} C_VEL
LIN {X 0,Y 515.152,Z 337.249,A -85,B 0,C 180,E1 -5468.336,E2 -5468.336} C_VEL
LIN {X 0,Y 514.593,Z 396.896,A -85,B 0,C 180,E1 -5469.228,E2 -5469.228} C_VEL
LIN {X 0,Y 513.848,Z 478.897,A -85,B 0,C 180,E1 -5470.451,E2 -5470.451} C_VEL
LIN {X 0,Y 513.579,Z 494.931,A -85,B 0,C 180,E1 -5470.773,E2 -5470.773} C_VEL
LIN {X 0,Y 513.184,Z 509.431,A -85,B 0,C 180,E1 -5471.215,E2 -5471.215} C_VEL
LIN {X 0,Y 512.692,Z 524.314,A -85,B 0,C 180,E1 -5471.83,E2 -5471.83} C_VEL
LIN {X 0,Y 512.198,Z 539.324,A -85,B 0,C 180,E1 -5472.638,E2 -5472.638} C_VEL
LIN {X 0,Y 511.636,Z 552.874,A -85,B 0,C 180,E1 -5473.543,E2 -5473.543} C_VEL
LIN {X 0,Y 511.175,Z 565.325,A -85,B 0,C 180,E1 -5474.552,E2 -5474.552} C_VEL
LIN {X 0,Y 510.639,Z 576.779,A -85,B 0,C 180,E1 -5475.658,E2 -5475.658} C_VEL
LIN {X 0,Y 510.281,Z 587.31,A -85,B 0,C 180,E1 -5476.866,E2 -5476.866} C_VEL
LIN {X 0,Y 509.889,Z 596.65,A -85,B 0,C 180,E1 -5478.132,E2 -5478.132} C_VEL
LIN {X 0,Y 509.733,Z 605.016,A -85,B 0,C 180,E1 -5479.475,E2 -5479.475} C_VEL
LIN {X 0,Y 509.471,Z 612.314,A -85,B 0,C 180,E1 -5480.873,E2 -5480.873} C_VEL
LIN {X 0,Y 509.326,Z 619.07,A -85,B 0,C 180,E1 -5482.469,E2 -5482.469} C_VEL
LIN {X 0,Y 509.271,Z 624.351,A -85,B 0,C 180,E1 -5484.06,E2 -5484.06} C_VEL
LIN {X 0,Y 509.158,Z 627.389,A -85,B 0,C 180,E1 -5485.251,E2 -5485.251} C_VEL
LIN {X 0,Y 509.189,Z 630.363,A -85,B 0,C 180,E1 -5486.836,E2 -5486.836} C_VEL
LIN {X 0,Y 509.11,Z 632.125,A -85,B 0,C 180,E1 -5488.419,E2 -5488.419} C_VEL
LIN {X 0,Y 509.066,Z 632.717,A -85,B 0,C 180,E1 -5490.001,E2 -5490.001} C_VEL
LIN {X 0,Y 509.11,Z 632.101,A -85,B 0,C 180,E1 -5491.583,E2 -5491.583} C_VEL
LIN {X 0,Y 509.19,Z 630.313,A -85,B 0,C 180,E1 -5493.166,E2 -5493.166} C_VEL
LIN {X 0,Y 509.159,Z 627.308,A -85,B 0,C 180,E1 -5494.752,E2 -5494.752} C_VEL
LIN {X 0,Y 509.265,Z 624.24,A -85,B 0,C 180,E1 -5495.942,E2 -5495.942} C_VEL
LIN {X 0,Y 509.339,Z 618.909,A -85,B 0,C 180,E1 -5497.533,E2 -5497.533} C_VEL
LIN {X 0,Y 509.473,Z 612.07,A -85,B 0,C 180,E1 -5499.129,E2 -5499.129} C_VEL
LIN {X 0,Y 509.734,Z 604.694,A -85,B 0,C 180,E1 -5500.527,E2 -5500.527} C_VEL
LIN {X 0,Y 509.925,Z 595.785,A -85,B 0,C 180,E1 -5501.932,E2 -5501.932} C_VEL
LIN {X 0,Y 510.316,Z 585.039,A -85,B 0,C 180,E1 -5503.338,E2 -5503.338} C_VEL
LIN {X 0,Y 510.724,Z 573.989,A -85,B 0,C 180,E1 -5504.546,E2 -5504.546} C_VEL
LIN {X 0,Y 511.167,Z 562.103,A -85,B 0,C 180,E1 -5505.638,E2 -5505.638} C_VEL
LIN {X 0,Y 511.629,Z 548.661,A -85,B 0,C 180,E1 -5506.664,E2 -5506.664} C_VEL
LIN {X 0,Y 512.235,Z 534.038,A -85,B 0,C 180,E1 -5507.569,E2 -5507.569} C_VEL
LIN {X 0,Y 512.693,Z 519.758,A -85,B 0,C 180,E1 -5508.275,E2 -5508.275} C_VEL
LIN {X 0,Y 513.089,Z 504.226,A -85,B 0,C 180,E1 -5508.865,E2 -5508.865} C_VEL
LIN {X 0,Y 513.456,Z 488.61,A -85,B 0,C 180,E1 -5509.283,E2 -5509.283} C_VEL
LIN {X 0,Y 513.66,Z 465.451,A -85,B 0,C 180,E1 -5509.664,E2 -5509.664} C_VEL
LIN {X 0,Y 514.669,Z 366.649,A -85,B 0,C 180,E1 -5511.167,E2 -5511.167} C_VEL
LIN {X 0,Y 514.939,Z 335.878,A -85,B 0,C 180,E1 -5511.663,E2 -5511.663} C_VEL
LIN {X 0,Y 511.854,Z 317.548,A -85,B 0,C 180,E1 -5512.113,E2 -5512.113} C_VEL
LIN {X 0,Y 512.545,Z 296.581,A -85,B 0,C 180,E1 -5514.723,E2 -5514.723} C_VEL
LIN {X 0,Y 513.295,Z 276.019,A -85,B 0,C 180,E1 -5517.354,E2 -5517.354} C_VEL
LIN {X 0,Y 512.788,Z 271.75,A -85,B 0,C 180,E1 -5517.952,E2 -5517.952} C_VEL
LIN {X 0,Y 509.87,Z 259.6,A -85,B 0,C 180,E1 -5519.808,E2 -5519.808} C_VEL
LIN {X 0,Y 509.878,Z 259.602,A -85,B 0,C 180,E1 -5522.774,E2 -5522.774} C_VEL
LIN {X 0,Y 509.831,Z 259.604,A -85,B 0,C 180,E1 -5525.579,E2 -5525.579} C_VEL
LIN {X 0,Y 509.856,Z 259.6,A -85,B 0,C 180,E1 -5528.338,E2 -5528.338} C_VEL
LIN {X 0,Y 509.861,Z 259.6,A -85,B 0,C 180,E1 -5531.426,E2 -5531.426} C_VEL
LIN {X 0,Y 509.863,Z 259.602,A -85,B 0,C 180,E1 -5534.668,E2 -5534.668} C_VEL
LIN {X 0,Y 509.861,Z 259.598,A -85,B 0,C 180,E1 -5538.104,E2 -5538.104} C_VEL
LIN {X 0,Y 509.851,Z 259.604,A -85,B 0,C 180,E1 -5540.648,E2 -5540.648} C_VEL
LIN {X 0,Y 509.815,Z 259.604,A -85,B 0,C 180,E1 -5543.646,E2 -5543.646} C_VEL
LIN {X 0,Y 509.865,Z 259.603,A -85,B 0,C 180,E1 -5546.539,E2 -5546.539} C_VEL
LIN {X 0,Y 509.851,Z 259.6,A -85,B 0,C 180,E1 -5549.334,E2 -5549.334} C_VEL
LIN {X 0,Y 509.854,Z 259.604,A -85,B 0,C 180,E1 -5552.052,E2 -5552.052} C_VEL
LIN {X 0,Y 509.843,Z 259.604,A -85,B 0,C 180,E1 -5554.702,E2 -5554.702} C_VEL
LIN {X 0,Y 509.885,Z 259.807,A -85,B 0,C 180,E1 -5556.331,E2 -5556.331} C_VEL
LIN {X 0,Y 511.83,Z 268.238,A -85,B 0,C 180,E1 -5557.983,E2 -5557.983} C_VEL
LIN {X 0,Y 513.945,Z 274.122,A -85,B 0,C 180,E1 -5558.187,E2 -5558.187} C_VEL
LIN {X 0,Y 515.387,Z 281.343,A -85,B 0,C 180,E1 -5558.382,E2 -5558.382} C_VEL
LIN {X 0,Y 513.894,Z 399.629,A -85,B 0,C 180,E1 -5560.241,E2 -5560.241} C_VEL
LIN {X 0,Y 513.607,Z 432.356,A -85,B 0,C 180,E1 -5560.755,E2 -5560.755} C_VEL
LIN {X 0,Y 513.367,Z 447.826,A -85,B 0,C 180,E1 -5561.157,E2 -5561.157} C_VEL
LIN {X 0,Y 513.026,Z 462.24,A -85,B 0,C 180,E1 -5561.686,E2 -5561.686} C_VEL
LIN {X 0,Y 512.605,Z 475.975,A -85,B 0,C 180,E1 -5562.341,E2 -5562.341} C_VEL
LIN {X 0,Y 512.18,Z 489.442,A -85,B 0,C 180,E1 -5563.149,E2 -5563.149} C_VEL
LIN {X 0,Y 511.651,Z 501.819,A -85,B 0,C 180,E1 -5564.054,E2 -5564.054} C_VEL
LIN {X 0,Y 511.155,Z 514.358,A -85,B 0,C 180,E1 -5565.162,E2 -5565.162} C_VEL
LIN {X 0,Y 510.773,Z 524.802,A -85,B 0,C 180,E1 -5566.269,E2 -5566.269} C_VEL
LIN {X 0,Y 510.303,Z 534.598,A -85,B 0,C 180,E1 -5567.492,E2 -5567.492} C_VEL
LIN {X 0,Y 510.011,Z 543.862,A -85,B 0,C 180,E1 -5568.876,E2 -5568.876} C_VEL
LIN {X 0,Y 509.703,Z 551.652,A -85,B 0,C 180,E1 -5570.275,E2 -5570.275} C_VEL
LIN {X 0,Y 509.501,Z 558.098,A -85,B 0,C 180,E1 -5571.672,E2 -5571.672} C_VEL
LIN {X 0,Y 509.395,Z 562.628,A -85,B 0,C 180,E1 -5572.867,E2 -5572.867} C_VEL
LIN {X 0,Y 509.318,Z 567.454,A -85,B 0,C 180,E1 -5574.456,E2 -5574.456} C_VEL
LIN {X 0,Y 509.255,Z 570.962,A -85,B 0,C 180,E1 -5576.043,E2 -5576.043} C_VEL
LIN {X 0,Y 509.19,Z 573.298,A -85,B 0,C 180,E1 -5577.626,E2 -5577.626} C_VEL
LIN {X 0,Y 509.076,Z 574.45,A -85,B 0,C 180,E1 -5579.208,E2 -5579.208} C_VEL
LIN {X 0,Y 509.076,Z 574.453,A -85,B 0,C 180,E1 -5580.79,E2 -5580.79} C_VEL
LIN {X 0,Y 509.191,Z 573.339,A -85,B 0,C 180,E1 -5582.372,E2 -5582.372} C_VEL
LIN {X 0,Y 509.255,Z 571.038,A -85,B 0,C 180,E1 -5583.956,E2 -5583.956} C_VEL
LIN {X 0,Y 509.311,Z 567.58,A -85,B 0,C 180,E1 -5585.542,E2 -5585.542} C_VEL
LIN {X 0,Y 509.37,Z 562.795,A -85,B 0,C 180,E1 -5587.133,E2 -5587.133} C_VEL
LIN {X 0,Y 509.543,Z 556.614,A -85,B 0,C 180,E1 -5588.726,E2 -5588.726} C_VEL
LIN {X 0,Y 509.749,Z 548.809,A -85,B 0,C 180,E1 -5590.324,E2 -5590.324} C_VEL
LIN {X 0,Y 510.049,Z 540.04,A -85,B 0,C 180,E1 -5591.792,E2 -5591.792} C_VEL
LIN {X 0,Y 510.468,Z 530.394,A -85,B 0,C 180,E1 -5593.13,E2 -5593.13} C_VEL
LIN {X 0,Y 510.925,Z 520.066,A -85,B 0,C 180,E1 -5594.335,E2 -5594.335} C_VEL
LIN {X 0,Y 511.408,Z 508.483,A -85,B 0,C 180,E1 -5595.471,E2 -5595.471} C_VEL
LIN {X 0,Y 511.937,Z 495.225,A -85,B 0,C 180,E1 -5596.55,E2 -5596.55} C_VEL
LIN {X 0,Y 512.498,Z 481.573,A -85,B 0,C 180,E1 -5597.455,E2 -5597.455} C_VEL
LIN {X 0,Y 512.933,Z 467.381,A -85,B 0,C 180,E1 -5598.213,E2 -5598.213} C_VEL
LIN {X 0,Y 513.336,Z 452.489,A -85,B 0,C 180,E1 -5598.828,E2 -5598.828} C_VEL
LIN {X 0,Y 513.706,Z 436.695,A -85,B 0,C 180,E1 -5599.297,E2 -5599.297} C_VEL
LIN {X 0,Y 513.917,Z 420.79,A -85,B 0,C 180,E1 -5599.6,E2 -5599.6} C_VEL
LIN {X 0,Y 515.287,Z 279.985,A -85,B 0,C 180,E1 -5601.729,E2 -5601.729} C_VEL
LIN {X 0,Y 512.814,Z 270.21,A -85,B 0,C 180,E1 -5601.996,E2 -5601.996} C_VEL
LIN {X 0,Y 511.142,Z 265.666,A -85,B 0,C 180,E1 -5602.151,E2 -5602.151} C_VEL
LIN {X 0,Y 509.833,Z 259.606,A -85,B 0,C 180,E1 -5603.266,E2 -5603.266} C_VEL
LIN {X 0,Y 509.876,Z 259.597,A -85,B 0,C 180,E1 -5606.369,E2 -5606.369} C_VEL
LIN {X 0,Y 509.851,Z 259.597,A -85,B 0,C 180,E1 -5608.845,E2 -5608.845} C_VEL
LIN {X 0,Y 509.835,Z 259.601,A -85,B 0,C 180,E1 -5610.148,E2 -5610.148} C_VEL
LIN {X 0,Y 509.164,Z 259.684,A -85,B 0,C 180,E1 -5610.807,E2 -5610.807} C_VEL
LIN {X 0,Y 506.316,Z 260.045,A -85,B 0,C 180,E1 -5611.877,E2 -5611.877} C_VEL
LIN {X 0,Y 503.911,Z 260.339,A -85,B 0,C 180,E1 -5612.739,E2 -5612.739} C_VEL
LIN {X 0,Y 502.881,Z 260.466,A -85,B 0,C 180,E1 -5613.405,E2 -5613.405} C_VEL
LIN {X 0,Y 502.797,Z 260.477,A -85,B 0,C 180,E1 -5613.63,E2 -5613.63} C_VEL
LIN {X 0,Y 502.767,Z 260.486,A -85,B 0,C 180,E1 -5615.951,E2 -5615.951} C_VEL
LIN {X 0,Y 502.799,Z 260.474,A -85,B 0,C 180,E1 -5618.975,E2 -5618.975} C_VEL
LIN {X 0,Y 502.802,Z 260.477,A -85,B 0,C 180,E1 -5622.198,E2 -5622.198} C_VEL
LIN {X 0,Y 502.784,Z 260.48,A -85,B 0,C 180,E1 -5625.469,E2 -5625.469} C_VEL
LIN {X 0,Y 502.817,Z 260.472,A -85,B 0,C 180,E1 -5628.933,E2 -5628.933} C_VEL
LIN {X 0,Y 502.79,Z 260.48,A -85,B 0,C 180,E1 -5632.045,E2 -5632.045} C_VEL
LIN {X 0,Y 502.792,Z 260.475,A -85,B 0,C 180,E1 -5635.033,E2 -5635.033} C_VEL
LIN {X 0,Y 502.778,Z 260.483,A -85,B 0,C 180,E1 -5637.914,E2 -5637.914} C_VEL
LIN {X 0,Y 502.809,Z 260.473,A -85,B 0,C 180,E1 -5640.71,E2 -5640.71} C_VEL
LIN {X 0,Y 502.84,Z 260.474,A -85,B 0,C 180,E1 -5643.442,E2 -5643.442} C_VEL
LIN {X 0,Y 502.769,Z 260.481,A -85,B 0,C 180,E1 -5646.084,E2 -5646.084} C_VEL
LIN {X 0,Y 502.777,Z 260.477,A -85,B 0,C 180,E1 -5648.688,E2 -5648.688} C_VEL
LIN {X 0,Y 502.82,Z 260.474,A -85,B 0,C 180,E1 -5651.247,E2 -5651.247} C_VEL
LIN {X 0,Y 502.842,Z 260.469,A -85,B 0,C 180,E1 -5654.599,E2 -5654.599} C_VEL
LIN {X 0,Y 502.869,Z 260.468,A -85,B 0,C 180,E1 -5658.038,E2 -5658.038} C_VEL
LIN {X 0,Y 502.866,Z 260.468,A -85,B 0,C 180,E1 -5661.156,E2 -5661.156} C_VEL
LIN {X 0,Y 502.897,Z 260.471,A -85,B 0,C 180,E1 -5663.58,E2 -5663.58} C_VEL
LIN {X 0,Y 502.888,Z 260.463,A -85,B 0,C 180,E1 -5666.794,E2 -5666.794} C_VEL
LIN {X 0,Y 503.027,Z 260.449,A -85,B 0,C 180,E1 -5669.198,E2 -5669.198} C_VEL
LIN {X 0,Y 502.895,Z 260.47,A -85,B 0,C 180,E1 -5671.601,E2 -5671.601} C_VEL
LIN {X 0,Y 502.889,Z 260.467,A -85,B 0,C 180,E1 -5673.203,E2 -5673.203} C_VEL
LIN {X 0,Y 502.896,Z 260.462,A -85,B 0,C 180,E1 -5676.418,E2 -5676.418} C_VEL
LIN {X 0,Y 502.86,Z 260.467,A -85,B 0,C 180,E1 -5678.842,E2 -5678.842} C_VEL
LIN {X 0,Y 502.835,Z 260.471,A -85,B 0,C 180,E1 -5682.101,E2 -5682.101} C_VEL
LIN {X 0,Y 502.837,Z 260.477,A -85,B 0,C 180,E1 -5685.399,E2 -5685.399} C_VEL
LIN {X 0,Y 502.829,Z 260.471,A -85,B 0,C 180,E1 -5688.119,E2 -5688.119} C_VEL
LIN {X 0,Y 502.817,Z 260.472,A -85,B 0,C 180,E1 -5690.535,E2 -5690.535} C_VEL
LIN {X 0,Y 502.775,Z 260.48,A -85,B 0,C 180,E1 -5693.04,E2 -5693.04} C_VEL
LIN {X 0,Y 502.809,Z 260.478,A -85,B 0,C 180,E1 -5695.676,E2 -5695.676} C_VEL
LIN {X 0,Y 502.827,Z 260.47,A -85,B 0,C 180,E1 -5698.372,E2 -5698.372} C_VEL
LIN {X 0,Y 502.783,Z 260.483,A -85,B 0,C 180,E1 -5701.499,E2 -5701.499} C_VEL
LIN {X 0,Y 502.792,Z 260.475,A -85,B 0,C 180,E1 -5704.444,E2 -5704.444} C_VEL
LIN {X 0,Y 502.766,Z 260.485,A -85,B 0,C 180,E1 -5707.178,E2 -5707.178} C_VEL
LIN {X 0,Y 502.774,Z 260.478,A -85,B 0,C 180,E1 -5710.015,E2 -5710.015} C_VEL
LIN {X 0,Y 502.788,Z 260.475,A -85,B 0,C 180,E1 -5712.199,E2 -5712.199} C_VEL
LIN {X 0,Y 502.786,Z 260.482,A -85,B 0,C 180,E1 -5715.468,E2 -5715.468} C_VEL
LIN {X 0,Y 502.815,Z 260.473,A -85,B 0,C 180,E1 -5717.864,E2 -5717.864} C_VEL
LIN {X 0,Y 502.787,Z 260.481,A -85,B 0,C 180,E1 -5721.024,E2 -5721.024} C_VEL
LIN {X 0,Y 502.768,Z 260.478,A -85,B 0,C 180,E1 -5724.167,E2 -5724.167} C_VEL
LIN {X 0,Y 502.818,Z 260.477,A -85,B 0,C 180,E1 -5726.993,E2 -5726.993} C_VEL
LIN {X 0,Y 502.799,Z 260.474,A -85,B 0,C 180,E1 -5730.065,E2 -5730.065} C_VEL
LIN {X 0,Y 502.818,Z 260.473,A -85,B 0,C 180,E1 -5732.533,E2 -5732.533} C_VEL
LIN {X 0,Y 502.811,Z 260.479,A -85,B 0,C 180,E1 -5735.299,E2 -5735.299} C_VEL
LIN {X 0,Y 502.765,Z 260.479,A -85,B 0,C 180,E1 -5737.827,E2 -5737.827} C_VEL
LIN {X 0,Y 502.81,Z 260.473,A -85,B 0,C 180,E1 -5740.4,E2 -5740.4} C_VEL
LIN {X 0,Y 502.819,Z 260.478,A -85,B 0,C 180,E1 -5742.932,E2 -5742.932} C_VEL
LIN {X 0,Y 502.829,Z 260.474,A -85,B 0,C 180,E1 -5745.43,E2 -5745.43} C_VEL
LIN {X 0,Y 502.862,Z 260.47,A -85,B 0,C 180,E1 -5748.717,E2 -5748.717} C_VEL
LIN {X 0,Y 502.886,Z 260.463,A -85,B 0,C 180,E1 -5751.967,E2 -5751.967} C_VEL
LIN {X 0,Y 502.919,Z 260.46,A -85,B 0,C 180,E1 -5754.387,E2 -5754.387} C_VEL
LIN {X 0,Y 503.009,Z 260.45,A -85,B 0,C 180,E1 -5757.598,E2 -5757.598} C_VEL
LIN {X 0,Y 503.01,Z 260.448,A -85,B 0,C 180,E1 -5760.001,E2 -5760.001} C_VEL
LIN {X 0,Y 503.01,Z 260.449,A -85,B 0,C 180,E1 -5762.403,E2 -5762.403} C_VEL
LIN {X 0,Y 502.92,Z 260.46,A -85,B 0,C 180,E1 -5765.614,E2 -5765.614} C_VEL
LIN {X 0,Y 502.889,Z 260.463,A -85,B 0,C 180,E1 -5768.034,E2 -5768.034} C_VEL
LIN {X 0,Y 502.866,Z 260.47,A -85,B 0,C 180,E1 -5771.284,E2 -5771.284} C_VEL
LIN {X 0,Y 502.833,Z 260.474,A -85,B 0,C 180,E1 -5774.572,E2 -5774.572} C_VEL
LIN {X 0,Y 502.844,Z 260.468,A -85,B 0,C 180,E1 -5777.908,E2 -5777.908} C_VEL
LIN {X 0,Y 502.817,Z 260.475,A -85,B 0,C 180,E1 -5780.537,E2 -5780.537} C_VEL
LIN {X 0,Y 502.78,Z 260.483,A -85,B 0,C 180,E1 -5783.042,E2 -5783.042} C_VEL
LIN {X 0,Y 502.827,Z 260.471,A -85,B 0,C 180,E1 -5785.677,E2 -5785.677} C_VEL
LIN {X 0,Y 502.829,Z 260.473,A -85,B 0,C 180,E1 -5788.374,E2 -5788.374} C_VEL
LIN {X 0,Y 502.782,Z 260.477,A -85,B 0,C 180,E1 -5791.5,E2 -5791.5} C_VEL
LIN {X 0,Y 502.795,Z 260.475,A -85,B 0,C 180,E1 -5793.995,E2 -5793.995} C_VEL
LIN {X 0,Y 502.768,Z 260.481,A -85,B 0,C 180,E1 -5797.179,E2 -5797.179} C_VEL
LIN {X 0,Y 502.779,Z 260.477,A -85,B 0,C 180,E1 -5800.016,E2 -5800.016} C_VEL
LIN {X 0,Y 502.795,Z 260.476,A -85,B 0,C 180,E1 -5802.2,E2 -5802.2} C_VEL
LIN {X 0,Y 502.778,Z 260.477,A -85,B 0,C 180,E1 -5805.471,E2 -5805.471} C_VEL
LIN {X 0,Y 502.813,Z 260.48,A -85,B 0,C 180,E1 -5808.935,E2 -5808.935} C_VEL
LIN {X 0,Y 502.784,Z 260.478,A -85,B 0,C 180,E1 -5812.047,E2 -5812.047} C_VEL
LIN {X 0,Y 502.792,Z 260.479,A -85,B 0,C 180,E1 -5815.035,E2 -5815.035} C_VEL
LIN {X 0,Y 502.778,Z 260.479,A -85,B 0,C 180,E1 -5817.917,E2 -5817.917} C_VEL
LIN {X 0,Y 502.836,Z 260.606,A -85,B 0,C 180,E1 -5819.734,E2 -5819.734} C_VEL
LIN {X 0,Y 506.707,Z 276.261,A -85,B 0,C 180,E1 -5822.067,E2 -5822.067} C_VEL
LIN {X 0,Y 506.807,Z 281.512,A -85,B 0,C 180,E1 -5822.768,E2 -5822.768} C_VEL
LIN {X 0,Y 505.873,Z 305.113,A -85,B 0,C 180,E1 -5825.807,E2 -5825.807} C_VEL
LIN {X 0,Y 505.3,Z 319.189,A -85,B 0,C 180,E1 -5827.592,E2 -5827.592} C_VEL
LIN {X 0,Y 508.487,Z 337.241,A -85,B 0,C 180,E1 -5828.042,E2 -5828.042} C_VEL
LIN {X 0,Y 507.896,Z 397.398,A -85,B 0,C 180,E1 -5828.968,E2 -5828.968} C_VEL
LIN {X 0,Y 506.946,Z 485.794,A -85,B 0,C 180,E1 -5830.33,E2 -5830.33} C_VEL
LIN {X 0,Y 506.593,Z 502.093,A -85,B 0,C 180,E1 -5830.746,E2 -5830.746} C_VEL
LIN {X 0,Y 506.175,Z 516.924,A -85,B 0,C 180,E1 -5831.29,E2 -5831.29} C_VEL
LIN {X 0,Y 505.586,Z 531.408,A -85,B 0,C 180,E1 -5831.985,E2 -5831.985} C_VEL
LIN {X 0,Y 505.056,Z 544.918,A -85,B 0,C 180,E1 -5832.802,E2 -5832.802} C_VEL
LIN {X 0,Y 504.485,Z 558.684,A -85,B 0,C 180,E1 -5833.823,E2 -5833.823} C_VEL
LIN {X 0,Y 503.935,Z 571.18,A -85,B 0,C 180,E1 -5834.946,E2 -5834.946} C_VEL
LIN {X 0,Y 503.403,Z 583.41,A -85,B 0,C 180,E1 -5836.272,E2 -5836.272} C_VEL
LIN {X 0,Y 502.994,Z 592.901,A -85,B 0,C 180,E1 -5837.494,E2 -5837.494} C_VEL
LIN {X 0,Y 502.707,Z 602.192,A -85,B 0,C 180,E1 -5838.918,E2 -5838.918} C_VEL
LIN {X 0,Y 502.416,Z 609.889,A -85,B 0,C 180,E1 -5840.338,E2 -5840.338} C_VEL
LIN {X 0,Y 502.282,Z 617.076,A -85,B 0,C 180,E1 -5841.958,E2 -5841.958} C_VEL
LIN {X 0,Y 502.185,Z 622.717,A -85,B 0,C 180,E1 -5843.573,E2 -5843.573} C_VEL
LIN {X 0,Y 502.081,Z 626.974,A -85,B 0,C 180,E1 -5845.183,E2 -5845.183} C_VEL
LIN {X 0,Y 502.11,Z 629.959,A -85,B 0,C 180,E1 -5846.792,E2 -5846.792} C_VEL
LIN {X 0,Y 502.034,Z 631.726,A -85,B 0,C 180,E1 -5848.397,E2 -5848.397} C_VEL
LIN {X 0,Y 501.981,Z 632.315,A -85,B 0,C 180,E1 -5850.001,E2 -5850.001} C_VEL
LIN {X 0,Y 502.034,Z 631.688,A -85,B 0,C 180,E1 -5851.605,E2 -5851.605} C_VEL
LIN {X 0,Y 502.11,Z 629.886,A -85,B 0,C 180,E1 -5853.211,E2 -5853.211} C_VEL
LIN {X 0,Y 502.081,Z 626.857,A -85,B 0,C 180,E1 -5854.819,E2 -5854.819} C_VEL
LIN {X 0,Y 502.167,Z 622.542,A -85,B 0,C 180,E1 -5856.43,E2 -5856.43} C_VEL
LIN {X 0,Y 502.284,Z 616.817,A -85,B 0,C 180,E1 -5858.044,E2 -5858.044} C_VEL
LIN {X 0,Y 502.416,Z 609.519,A -85,B 0,C 180,E1 -5859.664,E2 -5859.664} C_VEL
LIN {X 0,Y 502.696,Z 601.691,A -85,B 0,C 180,E1 -5861.084,E2 -5861.084} C_VEL
LIN {X 0,Y 502.979,Z 592.237,A -85,B 0,C 180,E1 -5862.509,E2 -5862.509} C_VEL
LIN {X 0,Y 503.361,Z 582.575,A -85,B 0,C 180,E1 -5863.732,E2 -5863.732} C_VEL
LIN {X 0,Y 503.832,Z 570.066,A -85,B 0,C 180,E1 -5865.059,E2 -5865.059} C_VEL
LIN {X 0,Y 504.38,Z 557.256,A -85,B 0,C 180,E1 -5866.182,E2 -5866.182} C_VEL
LIN {X 0,Y 504.862,Z 544.635,A -85,B 0,C 180,E1 -5867.103,E2 -5867.103} C_VEL
LIN {X 0,Y 505.353,Z 530.972,A -85,B 0,C 180,E1 -5867.921,E2 -5867.921} C_VEL
LIN {X 0,Y 505.91,Z 516.007,A -85,B 0,C 180,E1 -5868.634,E2 -5868.634} C_VEL
LIN {X 0,Y 506.395,Z 499.995,A -85,B 0,C 180,E1 -5869.206,E2 -5869.206} C_VEL
LIN {X 0,Y 506.693,Z 485.188,A -85,B 0,C 180,E1 -5869.577,E2 -5869.577} C_VEL
LIN {X 0,Y 508.277,Z 353.205,A -85,B 0,C 180,E1 -5871.659,E2 -5871.659} C_VEL
LIN {X 0,Y 508.303,Z 336.575,A -85,B 0,C 180,E1 -5871.945,E2 -5871.945} C_VEL
LIN {X 0,Y 505.028,Z 316.761,A -85,B 0,C 180,E1 -5872.471,E2 -5872.471} C_VEL
LIN {X 0,Y 505.991,Z 291.221,A -85,B 0,C 180,E1 -5875.726,E2 -5875.726} C_VEL
LIN {X 0,Y 506.515,Z 276.259,A -85,B 0,C 180,E1 -5877.699,E2 -5877.699} C_VEL
LIN {X 0,Y 503.625,Z 263.514,A -85,B 0,C 180,E1 -5879.646,E2 -5879.646} C_VEL
LIN {X 0,Y 502.825,Z 260.477,A -85,B 0,C 180,E1 -5880.167,E2 -5880.167} C_VEL
LIN {X 0,Y 502.837,Z 260.48,A -85,B 0,C 180,E1 -5883.032,E2 -5883.032} C_VEL
LIN {X 0,Y 502.778,Z 260.481,A -85,B 0,C 180,E1 -5885.952,E2 -5885.952} C_VEL
LIN {X 0,Y 502.807,Z 260.482,A -85,B 0,C 180,E1 -5888.976,E2 -5888.976} C_VEL
LIN {X 0,Y 502.8,Z 260.478,A -85,B 0,C 180,E1 -5892.14,E2 -5892.14} C_VEL
LIN {X 0,Y 502.807,Z 260.477,A -85,B 0,C 180,E1 -5895.469,E2 -5895.469} C_VEL
LIN {X 0,Y 502.826,Z 260.478,A -85,B 0,C 180,E1 -5898.934,E2 -5898.934} C_VEL
LIN {X 0,Y 502.796,Z 260.479,A -85,B 0,C 180,E1 -5902.046,E2 -5902.046} C_VEL
LIN {X 0,Y 502.803,Z 260.48,A -85,B 0,C 180,E1 -5905.034,E2 -5905.034} C_VEL
LIN {X 0,Y 502.789,Z 260.481,A -85,B 0,C 180,E1 -5907.915,E2 -5907.915} C_VEL
LIN {X 0,Y 502.819,Z 260.48,A -85,B 0,C 180,E1 -5910.711,E2 -5910.711} C_VEL
LIN {X 0,Y 502.853,Z 260.473,A -85,B 0,C 180,E1 -5913.443,E2 -5913.443} C_VEL
LIN {X 0,Y 502.845,Z 260.578,A -85,B 0,C 180,E1 -5915.952,E2 -5915.952} C_VEL
LIN {X 0,Y 504.764,Z 268.855,A -85,B 0,C 180,E1 -5917.626,E2 -5917.626} C_VEL
LIN {X 0,Y 507.49,Z 275.87,A -85,B 0,C 180,E1 -5917.905,E2 -5917.905} C_VEL
LIN {X 0,Y 508.839,Z 282.442,A -85,B 0,C 180,E1 -5918.089,E2 -5918.089} C_VEL
LIN {X 0,Y 507.188,Z 398.125,A -85,B 0,C 180,E1 -5919.969,E2 -5919.969} C_VEL
LIN {X 0,Y 506.802,Z 433.412,A -85,B 0,C 180,E1 -5920.538,E2 -5920.538} C_VEL
LIN {X 0,Y 506.563,Z 448.729,A -85,B 0,C 180,E1 -5920.95,E2 -5920.95} C_VEL
LIN {X 0,Y 506.19,Z 462.956,A -85,B 0,C 180,E1 -5921.482,E2 -5921.482} C_VEL
LIN {X 0,Y 505.739,Z 477.529,A -85,B 0,C 180,E1 -5922.198,E2 -5922.198} C_VEL
LIN {X 0,Y 505.257,Z 490.807,A -85,B 0,C 180,E1 -5923.016,E2 -5923.016} C_VEL
LIN {X 0,Y 504.677,Z 504.03,A -85,B 0,C 180,E1 -5924.014,E2 -5924.014} C_VEL
LIN {X 0,Y 504.217,Z 515.48,A -85,B 0,C 180,E1 -5925.056,E2 -5925.056} C_VEL
LIN {X 0,Y 503.748,Z 526.726,A -85,B 0,C 180,E1 -5926.28,E2 -5926.28} C_VEL
LIN {X 0,Y 503.284,Z 536.145,A -85,B 0,C 180,E1 -5927.499,E2 -5927.499} C_VEL
LIN {X 0,Y 502.985,Z 545.351,A -85,B 0,C 180,E1 -5928.923,E2 -5928.923} C_VEL
LIN {X 0,Y 502.645,Z 552.965,A -85,B 0,C 180,E1 -5930.34,E2 -5930.34} C_VEL
LIN {X 0,Y 502.409,Z 560.042,A -85,B 0,C 180,E1 -5931.958,E2 -5931.958} C_VEL
LIN {X 0,Y 502.279,Z 565.583,A -85,B 0,C 180,E1 -5933.572,E2 -5933.572} C_VEL
LIN {X 0,Y 502.11,Z 569.762,A -85,B 0,C 180,E1 -5935.182,E2 -5935.182} C_VEL
LIN {X 0,Y 502.185,Z 572.673,A -85,B 0,C 180,E1 -5936.79,E2 -5936.79} C_VEL
LIN {X 0,Y 502.036,Z 574.435,A -85,B 0,C 180,E1 -5938.395,E2 -5938.395} C_VEL
LIN {X 0,Y 501.986,Z 575.024,A -85,B 0,C 180,E1 -5939.999,E2 -5939.999} C_VEL
LIN {X 0,Y 502.035,Z 574.44,A -85,B 0,C 180,E1 -5941.604,E2 -5941.604} C_VEL
LIN {X 0,Y 502.171,Z 572.711,A -85,B 0,C 180,E1 -5943.208,E2 -5943.208} C_VEL
LIN {X 0,Y 502.101,Z 569.826,A -85,B 0,C 180,E1 -5944.817,E2 -5944.817} C_VEL
LIN {X 0,Y 502.257,Z 565.681,A -85,B 0,C 180,E1 -5946.427,E2 -5946.427} C_VEL
LIN {X 0,Y 502.406,Z 560.193,A -85,B 0,C 180,E1 -5948.041,E2 -5948.041} C_VEL
LIN {X 0,Y 502.61,Z 553.187,A -85,B 0,C 180,E1 -5949.659,E2 -5949.659} C_VEL
LIN {X 0,Y 502.926,Z 545.666,A -85,B 0,C 180,E1 -5951.077,E2 -5951.077} C_VEL
LIN {X 0,Y 503.277,Z 536.577,A -85,B 0,C 180,E1 -5952.5,E2 -5952.5} C_VEL
LIN {X 0,Y 503.74,Z 525.57,A -85,B 0,C 180,E1 -5953.925,E2 -5953.925} C_VEL
LIN {X 0,Y 504.23,Z 514.217,A -85,B 0,C 180,E1 -5955.149,E2 -5955.149} C_VEL
LIN {X 0,Y 504.847,Z 501.704,A -85,B 0,C 180,E1 -5956.269,E2 -5956.269} C_VEL
LIN {X 0,Y 505.321,Z 489.406,A -85,B 0,C 180,E1 -5957.189,E2 -5957.189} C_VEL
LIN {X 0,Y 505.89,Z 476.064,A -85,B 0,C 180,E1 -5958.004,E2 -5958.004} C_VEL
LIN {X 0,Y 506.299,Z 463.649,A -85,B 0,C 180,E1 -5958.618,E2 -5958.618} C_VEL
LIN {X 0,Y 506.662,Z 448.939,A -85,B 0,C 180,E1 -5959.189,E2 -5959.189} C_VEL
LIN {X 0,Y 506.999,Z 434.071,A -85,B 0,C 180,E1 -5959.602,E2 -5959.602} C_VEL
LIN {X 0,Y 507.215,Z 414.227,A -85,B 0,C 180,E1 -5959.947,E2 -5959.947} C_VEL
LIN {X 0,Y 508.697,Z 281.115,A -85,B 0,C 180,E1 -5962.004,E2 -5962.004} C_VEL
LIN {X 0,Y 506.366,Z 272.309,A -85,B 0,C 180,E1 -5962.255,E2 -5962.255} C_VEL
LIN {X 0,Y 504.003,Z 265.994,A -85,B 0,C 180,E1 -5962.474,E2 -5962.474} C_VEL
LIN {X 0,Y 502.796,Z 260.484,A -85,B 0,C 180,E1 -5963.503,E2 -5963.503} C_VEL
LIN {X 0,Y 502.836,Z 260.472,A -85,B 0,C 180,E1 -5966.567,E2 -5966.567} C_VEL
LIN {X 0,Y 502.815,Z 260.48,A -85,B 0,C 180,E1 -5969.934,E2 -5969.934} C_VEL
LIN {X 0,Y 502.832,Z 260.47,A -85,B 0,C 180,E1 -5973.03,E2 -5973.03} C_VEL
LIN {X 0,Y 502.797,Z 260.477,A -85,B 0,C 180,E1 -5973.63,E2 -5973.63} C_VEL
LIN {X 0,Y 502.124,Z 260.565,A -85,B 0,C 180,E1 -5974.299,E2 -5974.299} C_VEL
LIN {X 0,Y 499.239,Z 260.922,A -85,B 0,C 180,E1 -5975.384,E2 -5975.384} C_VEL
LIN {X 0,Y 496.809,Z 261.224,A -85,B 0,C 180,E1 -5976.259,E2 -5976.259} C_VEL
LIN {X 0,Y 495.78,Z 261.349,A -85,B 0,C 180,E1 -5976.934,E2 -5976.934} C_VEL
LIN {X 0,Y 495.704,Z 261.359,A -85,B 0,C 180,E1 -5977.163,E2 -5977.163} C_VEL
LIN {X 0,Y 495.757,Z 261.357,A -85,B 0,C 180,E1 -5980.046,E2 -5980.046} C_VEL
LIN {X 0,Y 495.716,Z 261.356,A -85,B 0,C 180,E1 -5982.883,E2 -5982.883} C_VEL
LIN {X 0,Y 495.726,Z 261.361,A -85,B 0,C 180,E1 -5985.997,E2 -5985.997} C_VEL
LIN {X 0,Y 495.763,Z 261.353,A -85,B 0,C 180,E1 -5989.299,E2 -5989.299} C_VEL
LIN {X 0,Y 495.725,Z 261.356,A -85,B 0,C 180,E1 -5992.437,E2 -5992.437} C_VEL
LIN {X 0,Y 495.768,Z 261.354,A -85,B 0,C 180,E1 -5995.455,E2 -5995.455} C_VEL
LIN {X 0,Y 495.751,Z 261.353,A -85,B 0,C 180,E1 -5998.362,E2 -5998.362} C_VEL
LIN {X 0,Y 495.751,Z 261.358,A -85,B 0,C 180,E1 -6001.513,E2 -6001.513} C_VEL
LIN {X 0,Y 495.757,Z 261.357,A -85,B 0,C 180,E1 -6003.929,E2 -6003.929} C_VEL
LIN {X 0,Y 495.753,Z 261.353,A -85,B 0,C 180,E1 -6007.138,E2 -6007.138} C_VEL
LIN {X 0,Y 495.765,Z 261.353,A -85,B 0,C 180,E1 -6010.108,E2 -6010.108} C_VEL
LIN {X 0,Y 495.759,Z 261.351,A -85,B 0,C 180,E1 -6012.679,E2 -6012.679} C_VEL
LIN {X 0,Y 495.783,Z 261.351,A -85,B 0,C 180,E1 -6015.216,E2 -6015.216} C_VEL
LIN {X 0,Y 495.844,Z 261.34,A -85,B 0,C 180,E1 -6018.554,E2 -6018.554} C_VEL
LIN {X 0,Y 495.865,Z 261.343,A -85,B 0,C 180,E1 -6021.851,E2 -6021.851} C_VEL
LIN {X 0,Y 495.88,Z 261.337,A -85,B 0,C 180,E1 -6024.305,E2 -6024.305} C_VEL
LIN {X 0,Y 495.983,Z 261.332,A -85,B 0,C 180,E1 -6027.563,E2 -6027.563} C_VEL
LIN {X 0,Y 495.986,Z 261.326,A -85,B 0,C 180,E1 -6029.999,E2 -6029.999} C_VEL
LIN {X 0,Y 495.982,Z 261.323,A -85,B 0,C 180,E1 -6032.435,E2 -6032.435} C_VEL
LIN {X 0,Y 495.878,Z 261.342,A -85,B 0,C 180,E1 -6035.692,E2 -6035.692} C_VEL
LIN {X 0,Y 495.861,Z 261.339,A -85,B 0,C 180,E1 -6038.147,E2 -6038.147} C_VEL
LIN {X 0,Y 495.84,Z 261.349,A -85,B 0,C 180,E1 -6041.444,E2 -6041.444} C_VEL
LIN {X 0,Y 495.778,Z 261.349,A -85,B 0,C 180,E1 -6044.782,E2 -6044.782} C_VEL
LIN {X 0,Y 495.77,Z 261.357,A -85,B 0,C 180,E1 -6047.318,E2 -6047.318} C_VEL
LIN {X 0,Y 495.759,Z 261.354,A -85,B 0,C 180,E1 -6049.889,E2 -6049.889} C_VEL
LIN {X 0,Y 495.746,Z 261.354,A -85,B 0,C 180,E1 -6052.86,E2 -6052.86} C_VEL
LIN {X 0,Y 495.767,Z 261.351,A -85,B 0,C 180,E1 -6056.068,E2 -6056.068} C_VEL
LIN {X 0,Y 495.758,Z 261.353,A -85,B 0,C 180,E1 -6058.814,E2 -6058.814} C_VEL
LIN {X 0,Y 495.745,Z 261.356,A -85,B 0,C 180,E1 -6061.725,E2 -6061.725} C_VEL
LIN {X 0,Y 495.761,Z 261.352,A -85,B 0,C 180,E1 -6064.694,E2 -6064.694} C_VEL
LIN {X 0,Y 495.717,Z 261.362,A -85,B 0,C 180,E1 -6067.561,E2 -6067.561} C_VEL
LIN {X 0,Y 495.752,Z 261.353,A -85,B 0,C 180,E1 -6070.699,E2 -6070.699} C_VEL
LIN {X 0,Y 495.72,Z 261.359,A -85,B 0,C 180,E1 -6073.695,E2 -6073.695} C_VEL
LIN {X 0,Y 495.719,Z 261.356,A -85,B 0,C 180,E1 -6076.304,E2 -6076.304} C_VEL
LIN {X 0,Y 495.751,Z 261.361,A -85,B 0,C 180,E1 -6079.3,E2 -6079.3} C_VEL
LIN {X 0,Y 495.715,Z 261.357,A -85,B 0,C 180,E1 -6082.438,E2 -6082.438} C_VEL
LIN {X 0,Y 495.769,Z 261.355,A -85,B 0,C 180,E1 -6085.457,E2 -6085.457} C_VEL
LIN {X 0,Y 495.743,Z 261.353,A -85,B 0,C 180,E1 -6088.364,E2 -6088.364} C_VEL
LIN {X 0,Y 495.772,Z 261.354,A -85,B 0,C 180,E1 -6091.507,E2 -6091.507} C_VEL
LIN {X 0,Y 495.775,Z 261.349,A -85,B 0,C 180,E1 -6093.932,E2 -6093.932} C_VEL
LIN {X 0,Y 495.745,Z 261.362,A -85,B 0,C 180,E1 -6097.139,E2 -6097.139} C_VEL
LIN {X 0,Y 495.763,Z 261.35,A -85,B 0,C 180,E1 -6100.11,E2 -6100.11} C_VEL
LIN {X 0,Y 495.771,Z 261.352,A -85,B 0,C 180,E1 -6102.682,E2 -6102.682} C_VEL
LIN {X 0,Y 495.775,Z 261.356,A -85,B 0,C 180,E1 -6105.217,E2 -6105.217} C_VEL
LIN {X 0,Y 495.837,Z 261.343,A -85,B 0,C 180,E1 -6108.555,E2 -6108.555} C_VEL
LIN {X 0,Y 495.858,Z 261.339,A -85,B 0,C 180,E1 -6111.853,E2 -6111.853} C_VEL
LIN {X 0,Y 495.875,Z 261.337,A -85,B 0,C 180,E1 -6114.307,E2 -6114.307} C_VEL
LIN {X 0,Y 495.978,Z 261.326,A -85,B 0,C 180,E1 -6117.564,E2 -6117.564} C_VEL
LIN {X 0,Y 495.982,Z 261.323,A -85,B 0,C 180,E1 -6120.001,E2 -6120.001} C_VEL
LIN {X 0,Y 495.979,Z 261.325,A -85,B 0,C 180,E1 -6122.437,E2 -6122.437} C_VEL
LIN {X 0,Y 495.876,Z 261.337,A -85,B 0,C 180,E1 -6125.694,E2 -6125.694} C_VEL
LIN {X 0,Y 495.861,Z 261.339,A -85,B 0,C 180,E1 -6128.149,E2 -6128.149} C_VEL
LIN {X 0,Y 495.84,Z 261.343,A -85,B 0,C 180,E1 -6131.446,E2 -6131.446} C_VEL
LIN {X 0,Y 495.778,Z 261.355,A -85,B 0,C 180,E1 -6134.784,E2 -6134.784} C_VEL
LIN {X 0,Y 495.77,Z 261.353,A -85,B 0,C 180,E1 -6137.32,E2 -6137.32} C_VEL
LIN {X 0,Y 495.766,Z 261.35,A -85,B 0,C 180,E1 -6139.891,E2 -6139.891} C_VEL
LIN {X 0,Y 495.749,Z 261.361,A -85,B 0,C 180,E1 -6142.862,E2 -6142.862} C_VEL
LIN {X 0,Y 495.779,Z 261.349,A -85,B 0,C 180,E1 -6146.069,E2 -6146.069} C_VEL
LIN {X 0,Y 495.762,Z 261.359,A -85,B 0,C 180,E1 -6148.816,E2 -6148.816} C_VEL
LIN {X 0,Y 495.745,Z 261.353,A -85,B 0,C 180,E1 -6151.726,E2 -6151.726} C_VEL
LIN {X 0,Y 495.761,Z 261.358,A -85,B 0,C 180,E1 -6154.695,E2 -6154.695} C_VEL
LIN {X 0,Y 495.719,Z 261.356,A -85,B 0,C 180,E1 -6157.563,E2 -6157.563} C_VEL
LIN {X 0,Y 495.758,Z 261.359,A -85,B 0,C 180,E1 -6160.701,E2 -6160.701} C_VEL
LIN {X 0,Y 495.72,Z 261.356,A -85,B 0,C 180,E1 -6164.003,E2 -6164.003} C_VEL
LIN {X 0,Y 495.718,Z 261.36,A -85,B 0,C 180,E1 -6167.118,E2 -6167.118} C_VEL
LIN {X 0,Y 495.752,Z 261.354,A -85,B 0,C 180,E1 -6169.954,E2 -6169.954} C_VEL
LIN {X 0,Y 495.713,Z 261.364,A -85,B 0,C 180,E1 -6172.556,E2 -6172.556} C_VEL
LIN {X 0,Y 495.771,Z 261.35,A -85,B 0,C 180,E1 -6175.458,E2 -6175.458} C_VEL
LIN {X 0,Y 495.75,Z 261.357,A -85,B 0,C 180,E1 -6178.365,E2 -6178.365} C_VEL
LIN {X 0,Y 495.764,Z 261.405,A -85,B 0,C 180,E1 -6179.424,E2 -6179.424} C_VEL
LIN {X 0,Y 499.858,Z 277.799,A -85,B 0,C 180,E1 -6181.902,E2 -6181.902} C_VEL
LIN {X 0,Y 500.13,Z 281.189,A -85,B 0,C 180,E1 -6182.374,E2 -6182.374} C_VEL
LIN {X 0,Y 499.088,Z 303.101,A -85,B 0,C 180,E1 -6185.234,E2 -6185.234} C_VEL
LIN {X 0,Y 498.458,Z 318.875,A -85,B 0,C 180,E1 -6187.268,E2 -6187.268} C_VEL
LIN {X 0,Y 501.921,Z 338.552,A -85,B 0,C 180,E1 -6187.766,E2 -6187.766} C_VEL
LIN {X 0,Y 501.137,Z 410.02,A -85,B 0,C 180,E1 -6188.886,E2 -6188.886} C_VEL
LIN {X 0,Y 500.181,Z 486.649,A -85,B 0,C 180,E1 -6190.107,E2 -6190.107} C_VEL
LIN {X 0,Y 499.763,Z 502.787,A -85,B 0,C 180,E1 -6190.537,E2 -6190.537} C_VEL
LIN {X 0,Y 499.282,Z 517.866,A -85,B 0,C 180,E1 -6191.111,E2 -6191.111} C_VEL
LIN {X 0,Y 498.675,Z 532.354,A -85,B 0,C 180,E1 -6191.833,E2 -6191.833} C_VEL
LIN {X 0,Y 498.102,Z 545.635,A -85,B 0,C 180,E1 -6192.66,E2 -6192.66} C_VEL
LIN {X 0,Y 497.533,Z 557.973,A -85,B 0,C 180,E1 -6193.591,E2 -6193.591} C_VEL
LIN {X 0,Y 496.965,Z 570.533,A -85,B 0,C 180,E1 -6194.73,E2 -6194.73} C_VEL
LIN {X 0,Y 496.406,Z 582.826,A -85,B 0,C 180,E1 -6196.075,E2 -6196.075} C_VEL
LIN {X 0,Y 495.965,Z 592.341,A -85,B 0,C 180,E1 -6197.313,E2 -6197.313} C_VEL
LIN {X 0,Y 495.662,Z 601.673,A -85,B 0,C 180,E1 -6198.759,E2 -6198.759} C_VEL
LIN {X 0,Y 495.336,Z 609.403,A -85,B 0,C 180,E1 -6200.198,E2 -6200.198} C_VEL
LIN {X 0,Y 495.209,Z 616.62,A -85,B 0,C 180,E1 -6201.842,E2 -6201.842} C_VEL
LIN {X 0,Y 495.088,Z 622.522,A -85,B 0,C 180,E1 -6203.557,E2 -6203.557} C_VEL
LIN {X 0,Y 495.005,Z 626.559,A -85,B 0,C 180,E1 -6205.114,E2 -6205.114} C_VEL
LIN {X 0,Y 495.031,Z 629.556,A -85,B 0,C 180,E1 -6206.746,E2 -6206.746} C_VEL
LIN {X 0,Y 494.961,Z 631.328,A -85,B 0,C 180,E1 -6208.374,E2 -6208.374} C_VEL
LIN {X 0,Y 494.899,Z 631.912,A -85,B 0,C 180,E1 -6210.001,E2 -6210.001} C_VEL
LIN {X 0,Y 494.961,Z 631.275,A -85,B 0,C 180,E1 -6211.628,E2 -6211.628} C_VEL
LIN {X 0,Y 495.032,Z 629.452,A -85,B 0,C 180,E1 -6213.257,E2 -6213.257} C_VEL
LIN {X 0,Y 495.006,Z 626.403,A -85,B 0,C 180,E1 -6214.888,E2 -6214.888} C_VEL
LIN {X 0,Y 495.084,Z 622.056,A -85,B 0,C 180,E1 -6216.522,E2 -6216.522} C_VEL
LIN {X 0,Y 495.212,Z 616.288,A -85,B 0,C 180,E1 -6218.16,E2 -6218.16} C_VEL
LIN {X 0,Y 495.332,Z 608.937,A -85,B 0,C 180,E1 -6219.804,E2 -6219.804} C_VEL
LIN {X 0,Y 495.645,Z 601.05,A -85,B 0,C 180,E1 -6221.244,E2 -6221.244} C_VEL
LIN {X 0,Y 495.941,Z 591.526,A -85,B 0,C 180,E1 -6222.69,E2 -6222.69} C_VEL
LIN {X 0,Y 496.341,Z 581.804,A -85,B 0,C 180,E1 -6223.93,E2 -6223.93} C_VEL
LIN {X 0,Y 496.806,Z 570.245,A -85,B 0,C 180,E1 -6225.172,E2 -6225.172} C_VEL
LIN {X 0,Y 497.39,Z 557.488,A -85,B 0,C 180,E1 -6226.316,E2 -6226.316} C_VEL
LIN {X 0,Y 497.964,Z 543.526,A -85,B 0,C 180,E1 -6227.347,E2 -6227.347} C_VEL
LIN {X 0,Y 498.56,Z 528.733,A -85,B 0,C 180,E1 -6228.227,E2 -6228.227} C_VEL
LIN {X 0,Y 499.074,Z 514.527,A -85,B 0,C 180,E1 -6228.899,E2 -6228.899} C_VEL
LIN {X 0,Y 499.56,Z 499.416,A -85,B 0,C 180,E1 -6229.442,E2 -6229.442} C_VEL
LIN {X 0,Y 499.944,Z 484.218,A -85,B 0,C 180,E1 -6229.825,E2 -6229.825} C_VEL
LIN {X 0,Y 501.585,Z 357.683,A -85,B 0,C 180,E1 -6231.881,E2 -6231.881} C_VEL
LIN {X 0,Y 501.755,Z 337.707,A -85,B 0,C 180,E1 -6232.23,E2 -6232.23} C_VEL
LIN {X 0,Y 498.163,Z 316.128,A -85,B 0,C 180,E1 -6232.828,E2 -6232.828} C_VEL
LIN {X 0,Y 499.275,Z 291.011,A -85,B 0,C 180,E1 -6236.098,E2 -6236.098} C_VEL
LIN {X 0,Y 499.698,Z 277.807,A -85,B 0,C 180,E1 -6237.882,E2 -6237.882} C_VEL
LIN {X 0,Y 497.16,Z 266.49,A -85,B 0,C 180,E1 -6239.656,E2 -6239.656} C_VEL
LIN {X 0,Y 495.781,Z 261.356,A -85,B 0,C 180,E1 -6240.534,E2 -6240.534} C_VEL
LIN {X 0,Y 495.764,Z 261.36,A -85,B 0,C 180,E1 -6243.565,E2 -6243.565} C_VEL
LIN {X 0,Y 495.733,Z 261.361,A -85,B 0,C 180,E1 -6246.544,E2 -6246.544} C_VEL
LIN {X 0,Y 495.762,Z 261.356,A -85,B 0,C 180,E1 -6249.638,E2 -6249.638} C_VEL
LIN {X 0,Y 495.743,Z 261.36,A -85,B 0,C 180,E1 -6252.507,E2 -6252.507} C_VEL
LIN {X 0,Y 495.755,Z 261.358,A -85,B 0,C 180,E1 -6255.14,E2 -6255.14} C_VEL
LIN {X 0,Y 495.762,Z 261.356,A -85,B 0,C 180,E1 -6258.219,E2 -6258.219} C_VEL
LIN {X 0,Y 495.755,Z 261.355,A -85,B 0,C 180,E1 -6261.408,E2 -6261.408} C_VEL
LIN {X 0,Y 495.751,Z 261.361,A -85,B 0,C 180,E1 -6264.462,E2 -6264.462} C_VEL
LIN {X 0,Y 495.774,Z 261.353,A -85,B 0,C 180,E1 -6267.406,E2 -6267.406} C_VEL
LIN {X 0,Y 495.769,Z 261.358,A -85,B 0,C 180,E1 -6270.253,E2 -6270.253} C_VEL
LIN {X 0,Y 495.786,Z 261.354,A -85,B 0,C 180,E1 -6273.261,E2 -6273.261} C_VEL
LIN {X 0,Y 495.781,Z 261.378,A -85,B 0,C 180,E1 -6275.55,E2 -6275.55} C_VEL
LIN {X 0,Y 497.752,Z 269.718,A -85,B 0,C 180,E1 -6277.271,E2 -6277.271} C_VEL
LIN {X 0,Y 501.415,Z 278.699,A -85,B 0,C 180,E1 -6277.642,E2 -6277.642} C_VEL
LIN {X 0,Y 502.319,Z 284.06,A -85,B 0,C 180,E1 -6277.79,E2 -6277.79} C_VEL
LIN {X 0,Y 500.536,Z 393.888,A -85,B 0,C 180,E1 -6279.637,E2 -6279.637} C_VEL
LIN {X 0,Y 500.077,Z 433.425,A -85,B 0,C 180,E1 -6280.288,E2 -6280.288} C_VEL
LIN {X 0,Y 499.775,Z 449.322,A -85,B 0,C 180,E1 -6280.72,E2 -6280.72} C_VEL
LIN {X 0,Y 499.374,Z 463.792,A -85,B 0,C 180,E1 -6281.273,E2 -6281.273} C_VEL
LIN {X 0,Y 498.95,Z 477.373,A -85,B 0,C 180,E1 -6281.947,E2 -6281.947} C_VEL
LIN {X 0,Y 498.448,Z 490.741,A -85,B 0,C 180,E1 -6282.776,E2 -6282.776} C_VEL
LIN {X 0,Y 497.855,Z 503.314,A -85,B 0,C 180,E1 -6283.726,E2 -6283.726} C_VEL
LIN {X 0,Y 497.319,Z 515.566,A -85,B 0,C 180,E1 -6284.844,E2 -6284.844} C_VEL
LIN {X 0,Y 496.82,Z 526.88,A -85,B 0,C 180,E1 -6286.085,E2 -6286.085} C_VEL
LIN {X 0,Y 496.252,Z 537.817,A -85,B 0,C 180,E1 -6287.527,E2 -6287.527} C_VEL
LIN {X 0,Y 495.94,Z 546.836,A -85,B 0,C 180,E1 -6288.97,E2 -6288.97} C_VEL
LIN {X 0,Y 495.572,Z 555.232,A -85,B 0,C 180,E1 -6290.613,E2 -6290.613} C_VEL
LIN {X 0,Y 495.319,Z 561.94,A -85,B 0,C 180,E1 -6292.253,E2 -6292.253} C_VEL
LIN {X 0,Y 495.22,Z 566.61,A -85,B 0,C 180,E1 -6293.697,E2 -6293.697} C_VEL
LIN {X 0,Y 495.037,Z 570.153,A -85,B 0,C 180,E1 -6295.113,E2 -6295.113} C_VEL
LIN {X 0,Y 495.102,Z 573.08,A -85,B 0,C 180,E1 -6296.744,E2 -6296.744} C_VEL
LIN {X 0,Y 494.963,Z 574.839,A -85,B 0,C 180,E1 -6298.372,E2 -6298.372} C_VEL
LIN {X 0,Y 494.903,Z 575.43,A -85,B 0,C 180,E1 -6299.999,E2 -6299.999} C_VEL
LIN {X 0,Y 494.962,Z 574.831,A -85,B 0,C 180,E1 -6301.627,E2 -6301.627} C_VEL
LIN {X 0,Y 495.09,Z 573.089,A -85,B 0,C 180,E1 -6303.254,E2 -6303.254} C_VEL
LIN {X 0,Y 495.027,Z 570.178,A -85,B 0,C 180,E1 -6304.886,E2 -6304.886} C_VEL
LIN {X 0,Y 495.205,Z 566.006,A -85,B 0,C 180,E1 -6306.519,E2 -6306.519} C_VEL
LIN {X 0,Y 495.35,Z 560.483,A -85,B 0,C 180,E1 -6308.156,E2 -6308.156} C_VEL
LIN {X 0,Y 495.591,Z 553.44,A -85,B 0,C 180,E1 -6309.797,E2 -6309.797} C_VEL
LIN {X 0,Y 495.916,Z 545.876,A -85,B 0,C 180,E1 -6311.236,E2 -6311.236} C_VEL
LIN {X 0,Y 496.313,Z 536.739,A -85,B 0,C 180,E1 -6312.678,E2 -6312.678} C_VEL
LIN {X 0,Y 496.801,Z 525.668,A -85,B 0,C 180,E1 -6314.124,E2 -6314.124} C_VEL
LIN {X 0,Y 497.331,Z 514.248,A -85,B 0,C 180,E1 -6315.364,E2 -6315.364} C_VEL
LIN {X 0,Y 497.957,Z 501.657,A -85,B 0,C 180,E1 -6316.5,E2 -6316.5} C_VEL
LIN {X 0,Y 498.504,Z 489.28,A -85,B 0,C 180,E1 -6317.432,E2 -6317.432} C_VEL
LIN {X 0,Y 499.069,Z 475.855,A -85,B 0,C 180,E1 -6318.259,E2 -6318.259} C_VEL
LIN {X 0,Y 499.613,Z 461.526,A -85,B 0,C 180,E1 -6318.96,E2 -6318.96} C_VEL
LIN {X 0,Y 500.002,Z 446.085,A -85,B 0,C 180,E1 -6319.535,E2 -6319.535} C_VEL
LIN {X 0,Y 500.356,Z 430.201,A -85,B 0,C 180,E1 -6319.94,E2 -6319.94} C_VEL
LIN {X 0,Y 502.099,Z 282.125,A -85,B 0,C 180,E1 -6322.288,E2 -6322.288} C_VEL
LIN {X 0,Y 499.966,Z 274.431,A -85,B 0,C 180,E1 -6322.516,E2 -6322.516} C_VEL
LIN {X 0,Y 496.833,Z 266.234,A -85,B 0,C 180,E1 -6322.825,E2 -6322.825} C_VEL
LIN {X 0,Y 495.735,Z 261.363,A -85,B 0,C 180,E1 -6323.747,E2 -6323.747} C_VEL
LIN {X 0,Y 495.761,Z 261.353,A -85,B 0,C 180,E1 -6326.976,E2 -6326.976} C_VEL
LIN {X 0,Y 495.764,Z 261.357,A -85,B 0,C 180,E1 -6330.146,E2 -6330.146} C_VEL
LIN {X 0,Y 495.793,Z 261.348,A -85,B 0,C 180,E1 -6333.243,E2 -6333.243} C_VEL
LIN {X 0,Y 495.711,Z 261.363,A -85,B 0,C 180,E1 -6336.086,E2 -6336.086} C_VEL
LIN {X 0,Y 495.704,Z 261.359,A -85,B 0,C 180,E1 -6337.163,E2 -6337.163} C_VEL
LIN {X 0,Y 495.062,Z 261.447,A -85,B 0,C 180,E1 -6337.841,E2 -6337.841} C_VEL
LIN {X 0,Y 492.234,Z 261.795,A -85,B 0,C 180,E1 -6338.943,E2 -6338.943} C_VEL
LIN {X 0,Y 489.824,Z 262.099,A -85,B 0,C 180,E1 -6339.83,E2 -6339.83} C_VEL
LIN {X 0,Y 488.778,Z 262.222,A -85,B 0,C 180,E1 -6340.515,E2 -6340.515} C_VEL
LIN {X 0,Y 488.688,Z 262.232,A -85,B 0,C 180,E1 -6340.747,E2 -6340.747} C_VEL
LIN {X 0,Y 488.689,Z 262.238,A -85,B 0,C 180,E1 -6344.022,E2 -6344.022} C_VEL
LIN {X 0,Y 488.683,Z 262.234,A -85,B 0,C 180,E1 -6347.175,E2 -6347.175} C_VEL
LIN {X 0,Y 488.731,Z 262.234,A -85,B 0,C 180,E1 -6349.675,E2 -6349.675} C_VEL
LIN {X 0,Y 488.676,Z 262.233,A -85,B 0,C 180,E1 -6352.84,E2 -6352.84} C_VEL
LIN {X 0,Y 488.72,Z 262.235,A -85,B 0,C 180,E1 -6355.885,E2 -6355.885} C_VEL
LIN {X 0,Y 488.687,Z 262.232,A -85,B 0,C 180,E1 -6358.819,E2 -6358.819} C_VEL
LIN {X 0,Y 488.708,Z 262.237,A -85,B 0,C 180,E1 -6361.668,E2 -6361.668} C_VEL
LIN {X 0,Y 488.711,Z 262.23,A -85,B 0,C 180,E1 -6364.441,E2 -6364.441} C_VEL
LIN {X 0,Y 488.716,Z 262.23,A -85,B 0,C 180,E1 -6367.152,E2 -6367.152} C_VEL
LIN {X 0,Y 488.719,Z 262.235,A -85,B 0,C 180,E1 -6369.809,E2 -6369.809} C_VEL
LIN {X 0,Y 488.709,Z 262.23,A -85,B 0,C 180,E1 -6372.422,E2 -6372.422} C_VEL
LIN {X 0,Y 488.755,Z 262.225,A -85,B 0,C 180,E1 -6374.998,E2 -6374.998} C_VEL
LIN {X 0,Y 488.798,Z 262.219,A -85,B 0,C 180,E1 -6378.386,E2 -6378.386} C_VEL
LIN {X 0,Y 488.81,Z 262.224,A -85,B 0,C 180,E1 -6381.732,E2 -6381.732} C_VEL
LIN {X 0,Y 488.838,Z 262.214,A -85,B 0,C 180,E1 -6384.223,E2 -6384.223} C_VEL
LIN {X 0,Y 488.95,Z 262.208,A -85,B 0,C 180,E1 -6387.527,E2 -6387.527} C_VEL
LIN {X 0,Y 488.958,Z 262.201,A -85,B 0,C 180,E1 -6389.999,E2 -6389.999} C_VEL
LIN {X 0,Y 488.95,Z 262.199,A -85,B 0,C 180,E1 -6392.47,E2 -6392.47} C_VEL
LIN {X 0,Y 488.837,Z 262.218,A -85,B 0,C 180,E1 -6395.775,E2 -6395.775} C_VEL
LIN {X 0,Y 488.806,Z 262.218,A -85,B 0,C 180,E1 -6398.265,E2 -6398.265} C_VEL
LIN {X 0,Y 488.794,Z 262.226,A -85,B 0,C 180,E1 -6401.611,E2 -6401.611} C_VEL
LIN {X 0,Y 488.75,Z 262.227,A -85,B 0,C 180,E1 -6404.999,E2 -6404.999} C_VEL
LIN {X 0,Y 488.743,Z 262.225,A -85,B 0,C 180,E1 -6408.441,E2 -6408.441} C_VEL
LIN {X 0,Y 488.694,Z 262.235,A -85,B 0,C 180,E1 -6411.07,E2 -6411.07} C_VEL
LIN {X 0,Y 488.667,Z 262.239,A -85,B 0,C 180,E1 -6413.745,E2 -6413.745} C_VEL
LIN {X 0,Y 488.779,Z 262.223,A -85,B 0,C 180,E1 -6416.943,E2 -6416.943} C_VEL
LIN {X 0,Y 488.696,Z 262.231,A -85,B 0,C 180,E1 -6420.362,E2 -6420.362} C_VEL
LIN {X 0,Y 488.722,Z 262.235,A -85,B 0,C 180,E1 -6423.484,E2 -6423.484} C_VEL
LIN {X 0,Y 488.673,Z 262.234,A -85,B 0,C 180,E1 -6426.355,E2 -6426.355} C_VEL
LIN {X 0,Y 488.687,Z 262.24,A -85,B 0,C 180,E1 -6429.254,E2 -6429.254} C_VEL
LIN {X 0,Y 488.709,Z 262.234,A -85,B 0,C 180,E1 -6431.602,E2 -6431.602} C_VEL
LIN {X 0,Y 488.697,Z 262.233,A -85,B 0,C 180,E1 -6434.801,E2 -6434.801} C_VEL
LIN {X 0,Y 488.704,Z 262.236,A -85,B 0,C 180,E1 -6437.477,E2 -6437.477} C_VEL
LIN {X 0,Y 488.718,Z 262.231,A -85,B 0,C 180,E1 -6439.676,E2 -6439.676} C_VEL
LIN {X 0,Y 488.666,Z 262.238,A -85,B 0,C 180,E1 -6442.841,E2 -6442.841} C_VEL
LIN {X 0,Y 488.719,Z 262.229,A -85,B 0,C 180,E1 -6445.887,E2 -6445.887} C_VEL
LIN {X 0,Y 488.679,Z 262.236,A -85,B 0,C 180,E1 -6448.82,E2 -6448.82} C_VEL
LIN {X 0,Y 488.729,Z 262.229,A -85,B 0,C 180,E1 -6451.671,E2 -6451.671} C_VEL
LIN {X 0,Y 488.732,Z 262.227,A -85,B 0,C 180,E1 -6454.444,E2 -6454.444} C_VEL
LIN {X 0,Y 488.707,Z 262.238,A -85,B 0,C 180,E1 -6457.153,E2 -6457.153} C_VEL
LIN {X 0,Y 488.714,Z 262.23,A -85,B 0,C 180,E1 -6459.811,E2 -6459.811} C_VEL
LIN {X 0,Y 488.719,Z 262.229,A -85,B 0,C 180,E1 -6462.424,E2 -6462.424} C_VEL
LIN {X 0,Y 488.747,Z 262.232,A -85,B 0,C 180,E1 -6465,E2 -6465} C_VEL
LIN {X 0,Y 488.791,Z 262.22,A -85,B 0,C 180,E1 -6468.388,E2 -6468.388} C_VEL
LIN {X 0,Y 488.802,Z 262.219,A -85,B 0,C 180,E1 -6471.734,E2 -6471.734} C_VEL
LIN {X 0,Y 488.833,Z 262.214,A -85,B 0,C 180,E1 -6474.225,E2 -6474.225} C_VEL
LIN {X 0,Y 488.946,Z 262.202,A -85,B 0,C 180,E1 -6477.529,E2 -6477.529} C_VEL
LIN {X 0,Y 488.963,Z 262.203,A -85,B 0,C 180,E1 -6480.824,E2 -6480.824} C_VEL
LIN {X 0,Y 488.947,Z 262.202,A -85,B 0,C 180,E1 -6482.472,E2 -6482.472} C_VEL
LIN {X 0,Y 488.834,Z 262.214,A -85,B 0,C 180,E1 -6485.777,E2 -6485.777} C_VEL
LIN {X 0,Y 488.805,Z 262.218,A -85,B 0,C 180,E1 -6488.267,E2 -6488.267} C_VEL
LIN {X 0,Y 488.794,Z 262.22,A -85,B 0,C 180,E1 -6491.613,E2 -6491.613} C_VEL
LIN {X 0,Y 488.75,Z 262.232,A -85,B 0,C 180,E1 -6495.001,E2 -6495.001} C_VEL
LIN {X 0,Y 488.744,Z 262.227,A -85,B 0,C 180,E1 -6498.443,E2 -6498.443} C_VEL
LIN {X 0,Y 488.696,Z 262.237,A -85,B 0,C 180,E1 -6501.072,E2 -6501.072} C_VEL
LIN {X 0,Y 488.677,Z 262.233,A -85,B 0,C 180,E1 -6503.747,E2 -6503.747} C_VEL
LIN {X 0,Y 488.781,Z 262.228,A -85,B 0,C 180,E1 -6506.945,E2 -6506.945} C_VEL
LIN {X 0,Y 488.699,Z 262.233,A -85,B 0,C 180,E1 -6510.364,E2 -6510.364} C_VEL
LIN {X 0,Y 488.725,Z 262.228,A -85,B 0,C 180,E1 -6513.485,E2 -6513.485} C_VEL
LIN {X 0,Y 488.673,Z 262.236,A -85,B 0,C 180,E1 -6516.356,E2 -6516.356} C_VEL
LIN {X 0,Y 488.692,Z 262.234,A -85,B 0,C 180,E1 -6519.256,E2 -6519.256} C_VEL
LIN {X 0,Y 488.699,Z 262.231,A -85,B 0,C 180,E1 -6521.601,E2 -6521.601} C_VEL
LIN {X 0,Y 488.693,Z 262.239,A -85,B 0,C 180,E1 -6524.804,E2 -6524.804} C_VEL
LIN {X 0,Y 488.685,Z 262.233,A -85,B 0,C 180,E1 -6527.476,E2 -6527.476} C_VEL
LIN {X 0,Y 488.726,Z 262.229,A -85,B 0,C 180,E1 -6529.678,E2 -6529.678} C_VEL
LIN {X 0,Y 488.664,Z 262.241,A -85,B 0,C 180,E1 -6532.842,E2 -6532.842} C_VEL
LIN {X 0,Y 488.724,Z 262.228,A -85,B 0,C 180,E1 -6535.888,E2 -6535.888} C_VEL
LIN {X 0,Y 488.749,Z 262.415,A -85,B 0,C 180,E1 -6539.138,E2 -6539.138} C_VEL
LIN {X 0,Y 492.929,Z 279.13,A -85,B 0,C 180,E1 -6541.703,E2 -6541.703} C_VEL
LIN {X 0,Y 493.339,Z 282.611,A -85,B 0,C 180,E1 -6542.2,E2 -6542.2} C_VEL
LIN {X 0,Y 492.251,Z 304.446,A -85,B 0,C 180,E1 -6545.092,E2 -6545.092} C_VEL
LIN {X 0,Y 491.643,Z 318.6,A -85,B 0,C 180,E1 -6546.943,E2 -6546.943} C_VEL
LIN {X 0,Y 495.344,Z 339.513,A -85,B 0,C 180,E1 -6547.477,E2 -6547.477} C_VEL
LIN {X 0,Y 493.436,Z 486.283,A -85,B 0,C 180,E1 -6549.85,E2 -6549.85} C_VEL
LIN {X 0,Y 493.004,Z 502.171,A -85,B 0,C 180,E1 -6550.279,E2 -6550.279} C_VEL
LIN {X 0,Y 492.481,Z 516.891,A -85,B 0,C 180,E1 -6550.84,E2 -6550.84} C_VEL
LIN {X 0,Y 491.934,Z 529.622,A -85,B 0,C 180,E1 -6551.467,E2 -6551.467} C_VEL
LIN {X 0,Y 491.287,Z 543.311,A -85,B 0,C 180,E1 -6552.304,E2 -6552.304} C_VEL
LIN {X 0,Y 490.699,Z 555.945,A -85,B 0,C 180,E1 -6553.249,E2 -6553.249} C_VEL
LIN {X 0,Y 490.146,Z 567.704,A -85,B 0,C 180,E1 -6554.299,E2 -6554.299} C_VEL
LIN {X 0,Y 489.525,Z 578.632,A -85,B 0,C 180,E1 -6555.45,E2 -6555.45} C_VEL
LIN {X 0,Y 489.117,Z 588.747,A -85,B 0,C 180,E1 -6556.71,E2 -6556.71} C_VEL
LIN {X 0,Y 488.617,Z 598.25,A -85,B 0,C 180,E1 -6558.112,E2 -6558.112} C_VEL
LIN {X 0,Y 488.431,Z 606.858,A -85,B 0,C 180,E1 -6559.64,E2 -6559.64} C_VEL
LIN {X 0,Y 488.139,Z 614.509,A -85,B 0,C 180,E1 -6561.306,E2 -6561.306} C_VEL
LIN {X 0,Y 488.048,Z 620.58,A -85,B 0,C 180,E1 -6562.97,E2 -6562.97} C_VEL
LIN {X 0,Y 487.997,Z 624.167,A -85,B 0,C 180,E1 -6564.215,E2 -6564.215} C_VEL
LIN {X 0,Y 487.928,Z 627.805,A -85,B 0,C 180,E1 -6565.871,E2 -6565.871} C_VEL
LIN {X 0,Y 487.955,Z 630.193,A -85,B 0,C 180,E1 -6567.525,E2 -6567.525} C_VEL
LIN {X 0,Y 487.832,Z 631.37,A -85,B 0,C 180,E1 -6569.176,E2 -6569.176} C_VEL
LIN {X 0,Y 487.832,Z 631.335,A -85,B 0,C 180,E1 -6570.827,E2 -6570.827} C_VEL
LIN {X 0,Y 487.985,Z 630.095,A -85,B 0,C 180,E1 -6572.477,E2 -6572.477} C_VEL
LIN {X 0,Y 487.932,Z 627.638,A -85,B 0,C 180,E1 -6574.131,E2 -6574.131} C_VEL
LIN {X 0,Y 488.015,Z 623.925,A -85,B 0,C 180,E1 -6575.787,E2 -6575.787} C_VEL
LIN {X 0,Y 488.065,Z 618.844,A -85,B 0,C 180,E1 -6577.447,E2 -6577.447} C_VEL
LIN {X 0,Y 488.203,Z 612.258,A -85,B 0,C 180,E1 -6579.112,E2 -6579.112} C_VEL
LIN {X 0,Y 488.474,Z 605.145,A -85,B 0,C 180,E1 -6580.571,E2 -6580.571} C_VEL
LIN {X 0,Y 488.73,Z 595.663,A -85,B 0,C 180,E1 -6582.166,E2 -6582.166} C_VEL
LIN {X 0,Y 489.108,Z 586.126,A -85,B 0,C 180,E1 -6583.504,E2 -6583.504} C_VEL
LIN {X 0,Y 489.646,Z 574.475,A -85,B 0,C 180,E1 -6584.867,E2 -6584.867} C_VEL
LIN {X 0,Y 490.152,Z 562.948,A -85,B 0,C 180,E1 -6586.001,E2 -6586.001} C_VEL
LIN {X 0,Y 490.697,Z 549.881,A -85,B 0,C 180,E1 -6587.075,E2 -6587.075} C_VEL
LIN {X 0,Y 491.4,Z 535.874,A -85,B 0,C 180,E1 -6588.017,E2 -6588.017} C_VEL
LIN {X 0,Y 491.984,Z 521.36,A -85,B 0,C 180,E1 -6588.803,E2 -6588.803} C_VEL
LIN {X 0,Y 492.493,Z 507.253,A -85,B 0,C 180,E1 -6589.404,E2 -6589.404} C_VEL
LIN {X 0,Y 492.958,Z 491.498,A -85,B 0,C 180,E1 -6589.899,E2 -6589.899} C_VEL
LIN {X 0,Y 493.32,Z 474.64,A -85,B 0,C 180,E1 -6590.239,E2 -6590.239} C_VEL
LIN {X 0,Y 494.703,Z 376.866,A -85,B 0,C 180,E1 -6591.855,E2 -6591.855} C_VEL
LIN {X 0,Y 495.209,Z 338.79,A -85,B 0,C 180,E1 -6592.532,E2 -6592.532} C_VEL
LIN {X 0,Y 491.372,Z 315.611,A -85,B 0,C 180,E1 -6593.19,E2 -6593.19} C_VEL
LIN {X 0,Y 492.535,Z 290.862,A -85,B 0,C 180,E1 -6596.482,E2 -6596.482} C_VEL
LIN {X 0,Y 493.011,Z 280.637,A -85,B 0,C 180,E1 -6597.892,E2 -6597.892} C_VEL
LIN {X 0,Y 491.167,Z 271.434,A -85,B 0,C 180,E1 -6599.346,E2 -6599.346} C_VEL
LIN {X 0,Y 488.726,Z 262.235,A -85,B 0,C 180,E1 -6600.937,E2 -6600.937} C_VEL
LIN {X 0,Y 488.735,Z 262.233,A -85,B 0,C 180,E1 -6604.113,E2 -6604.113} C_VEL
LIN {X 0,Y 488.685,Z 262.241,A -85,B 0,C 180,E1 -6607.159,E2 -6607.159} C_VEL
LIN {X 0,Y 488.724,Z 262.233,A -85,B 0,C 180,E1 -6610.345,E2 -6610.345} C_VEL
LIN {X 0,Y 488.692,Z 262.236,A -85,B 0,C 180,E1 -6613.655,E2 -6613.655} C_VEL
LIN {X 0,Y 488.693,Z 262.238,A -85,B 0,C 180,E1 -6616.346,E2 -6616.346} C_VEL
LIN {X 0,Y 488.739,Z 262.228,A -85,B 0,C 180,E1 -6619.677,E2 -6619.677} C_VEL
LIN {X 0,Y 488.676,Z 262.241,A -85,B 0,C 180,E1 -6622.84,E2 -6622.84} C_VEL
LIN {X 0,Y 488.736,Z 262.232,A -85,B 0,C 180,E1 -6625.887,E2 -6625.887} C_VEL
LIN {X 0,Y 488.698,Z 262.238,A -85,B 0,C 180,E1 -6628.82,E2 -6628.82} C_VEL
LIN {X 0,Y 488.719,Z 262.234,A -85,B 0,C 180,E1 -6631.669,E2 -6631.669} C_VEL
LIN {X 0,Y 488.729,Z 262.235,A -85,B 0,C 180,E1 -6634.443,E2 -6634.443} C_VEL
LIN {X 0,Y 488.74,Z 262.376,A -85,B 0,C 180,E1 -6635.154,E2 -6635.154} C_VEL
LIN {X 0,Y 490.782,Z 270.638,A -85,B 0,C 180,E1 -6636.891,E2 -6636.891} C_VEL
LIN {X 0,Y 495.301,Z 281.429,A -85,B 0,C 180,E1 -6637.362,E2 -6637.362} C_VEL
LIN {X 0,Y 495.883,Z 284.525,A -85,B 0,C 180,E1 -6637.455,E2 -6637.455} C_VEL
LIN {X 0,Y 493.889,Z 390.327,A -85,B 0,C 180,E1 -6639.296,E2 -6639.296} C_VEL
LIN {X 0,Y 493.358,Z 434.655,A -85,B 0,C 180,E1 -6640.053,E2 -6640.053} C_VEL
LIN {X 0,Y 493.017,Z 450.504,A -85,B 0,C 180,E1 -6640.499,E2 -6640.499} C_VEL
LIN {X 0,Y 492.546,Z 465.876,A -85,B 0,C 180,E1 -6641.111,E2 -6641.111} C_VEL
LIN {X 0,Y 492.021,Z 480.85,A -85,B 0,C 180,E1 -6641.9,E2 -6641.9} C_VEL
LIN {X 0,Y 491.406,Z 495.067,A -85,B 0,C 180,E1 -6642.843,E2 -6642.843} C_VEL
LIN {X 0,Y 490.828,Z 507.5,A -85,B 0,C 180,E1 -6643.853,E2 -6643.853} C_VEL
LIN {X 0,Y 490.216,Z 519.675,A -85,B 0,C 180,E1 -6645.045,E2 -6645.045} C_VEL
LIN {X 0,Y 489.713,Z 530.38,A -85,B 0,C 180,E1 -6646.302,E2 -6646.302} C_VEL
LIN {X 0,Y 489.204,Z 540.121,A -85,B 0,C 180,E1 -6647.663,E2 -6647.663} C_VEL
LIN {X 0,Y 488.797,Z 549.365,A -85,B 0,C 180,E1 -6649.227,E2 -6649.227} C_VEL
LIN {X 0,Y 488.456,Z 557.367,A -85,B 0,C 180,E1 -6650.893,E2 -6650.893} C_VEL
LIN {X 0,Y 488.246,Z 563.715,A -85,B 0,C 180,E1 -6652.556,E2 -6652.556} C_VEL
LIN {X 0,Y 488.145,Z 568.599,A -85,B 0,C 180,E1 -6654.215,E2 -6654.215} C_VEL
LIN {X 0,Y 488.053,Z 572.165,A -85,B 0,C 180,E1 -6655.871,E2 -6655.871} C_VEL
LIN {X 0,Y 487.997,Z 574.51,A -85,B 0,C 180,E1 -6657.523,E2 -6657.523} C_VEL
LIN {X 0,Y 487.836,Z 575.696,A -85,B 0,C 180,E1 -6659.174,E2 -6659.174} C_VEL
LIN {X 0,Y 487.836,Z 575.675,A -85,B 0,C 180,E1 -6660.825,E2 -6660.825} C_VEL
LIN {X 0,Y 487.996,Z 574.492,A -85,B 0,C 180,E1 -6662.476,E2 -6662.476} C_VEL
LIN {X 0,Y 488.051,Z 572.154,A -85,B 0,C 180,E1 -6664.128,E2 -6664.128} C_VEL
LIN {X 0,Y 488.133,Z 568.595,A -85,B 0,C 180,E1 -6665.784,E2 -6665.784} C_VEL
LIN {X 0,Y 488.215,Z 563.736,A -85,B 0,C 180,E1 -6667.443,E2 -6667.443} C_VEL
LIN {X 0,Y 488.425,Z 557.439,A -85,B 0,C 180,E1 -6669.106,E2 -6669.106} C_VEL
LIN {X 0,Y 488.747,Z 549.509,A -85,B 0,C 180,E1 -6670.773,E2 -6670.773} C_VEL
LIN {X 0,Y 489.136,Z 540.608,A -85,B 0,C 180,E1 -6672.3,E2 -6672.3} C_VEL
LIN {X 0,Y 489.626,Z 530.786,A -85,B 0,C 180,E1 -6673.699,E2 -6673.699} C_VEL
LIN {X 0,Y 490.165,Z 520.285,A -85,B 0,C 180,E1 -6674.956,E2 -6674.956} C_VEL
LIN {X 0,Y 490.793,Z 508.426,A -85,B 0,C 180,E1 -6676.144,E2 -6676.144} C_VEL
LIN {X 0,Y 491.357,Z 496.383,A -85,B 0,C 180,E1 -6677.157,E2 -6677.157} C_VEL
LIN {X 0,Y 492.022,Z 482.736,A -85,B 0,C 180,E1 -6678.099,E2 -6678.099} C_VEL
LIN {X 0,Y 492.521,Z 468.579,A -85,B 0,C 180,E1 -6678.888,E2 -6678.888} C_VEL
LIN {X 0,Y 493.029,Z 453.188,A -85,B 0,C 180,E1 -6679.548,E2 -6679.548} C_VEL
LIN {X 0,Y 493.448,Z 438.262,A -85,B 0,C 180,E1 -6680.014,E2 -6680.014} C_VEL
LIN {X 0,Y 493.711,Z 421.256,A -85,B 0,C 180,E1 -6680.356,E2 -6680.356} C_VEL
LIN {X 0,Y 495.478,Z 283.285,A -85,B 0,C 180,E1 -6682.575,E2 -6682.575} C_VEL
LIN {X 0,Y 493.747,Z 277.161,A -85,B 0,C 180,E1 -6682.761,E2 -6682.761} C_VEL
LIN {X 0,Y 489.672,Z 266.599,A -85,B 0,C 180,E1 -6683.159,E2 -6683.159} C_VEL
LIN {X 0,Y 488.712,Z 262.238,A -85,B 0,C 180,E1 -6683.997,E2 -6683.997} C_VEL
LIN {X 0,Y 488.726,Z 262.229,A -85,B 0,C 180,E1 -6686.927,E2 -6686.927} C_VEL
LIN {X 0,Y 488.723,Z 262.233,A -85,B 0,C 180,E1 -6690.218,E2 -6690.218} C_VEL
LIN {X 0,Y 488.734,Z 262.229,A -85,B 0,C 180,E1 -6693.483,E2 -6693.483} C_VEL
LIN {X 0,Y 488.672,Z 262.236,A -85,B 0,C 180,E1 -6696.352,E2 -6696.352} C_VEL
LIN {X 0,Y 488.699,Z 262.232,A -85,B 0,C 180,E1 -6699.253,E2 -6699.253} C_VEL
LIN {X 0,Y 488.688,Z 262.232,A -85,B 0,C 180,E1 -6700.747,E2 -6700.747} C_VEL
LIN {X 0,Y 488.008,Z 262.321,A -85,B 0,C 180,E1 -6701.435,E2 -6701.435} C_VEL
LIN {X 0,Y 485.152,Z 262.677,A -85,B 0,C 180,E1 -6702.553,E2 -6702.553} C_VEL
LIN {X 0,Y 482.752,Z 262.977,A -85,B 0,C 180,E1 -6703.453,E2 -6703.453} C_VEL
LIN {X 0,Y 481.73,Z 263.103,A -85,B 0,C 180,E1 -6704.149,E2 -6704.149} C_VEL
LIN {X 0,Y 481.651,Z 263.11,A -85,B 0,C 180,E1 -6704.385,E2 -6704.385} C_VEL
LIN {X 0,Y 481.629,Z 263.111,A -85,B 0,C 180,E1 -6706.852,E2 -6706.852} C_VEL
LIN {X 0,Y 481.674,Z 263.11,A -85,B 0,C 180,E1 -6710.058,E2 -6710.058} C_VEL
LIN {X 0,Y 481.622,Z 263.114,A -85,B 0,C 180,E1 -6713.252,E2 -6713.252} C_VEL
LIN {X 0,Y 481.673,Z 263.107,A -85,B 0,C 180,E1 -6716.326,E2 -6716.326} C_VEL
LIN {X 0,Y 481.646,Z 263.113,A -85,B 0,C 180,E1 -6719.416,E2 -6719.416} C_VEL
LIN {X 0,Y 481.664,Z 263.11,A -85,B 0,C 180,E1 -6722.165,E2 -6722.165} C_VEL
LIN {X 0,Y 481.684,Z 263.105,A -85,B 0,C 180,E1 -6724.967,E2 -6724.967} C_VEL
LIN {X 0,Y 481.644,Z 263.118,A -85,B 0,C 180,E1 -6727.703,E2 -6727.703} C_VEL
LIN {X 0,Y 481.698,Z 263.103,A -85,B 0,C 180,E1 -6730.392,E2 -6730.392} C_VEL
LIN {X 0,Y 481.674,Z 263.107,A -85,B 0,C 180,E1 -6733.032,E2 -6733.032} C_VEL
LIN {X 0,Y 481.683,Z 263.113,A -85,B 0,C 180,E1 -6735.637,E2 -6735.637} C_VEL
LIN {X 0,Y 481.744,Z 263.098,A -85,B 0,C 180,E1 -6738.214,E2 -6738.214} C_VEL
LIN {X 0,Y 481.755,Z 263.104,A -85,B 0,C 180,E1 -6741.611,E2 -6741.611} C_VEL
LIN {X 0,Y 481.799,Z 263.092,A -85,B 0,C 180,E1 -6744.138,E2 -6744.138} C_VEL
LIN {X 0,Y 481.917,Z 263.083,A -85,B 0,C 180,E1 -6747.491,E2 -6747.491} C_VEL
LIN {X 0,Y 481.897,Z 263.079,A -85,B 0,C 180,E1 -6750.834,E2 -6750.834} C_VEL
LIN {X 0,Y 481.917,Z 263.075,A -85,B 0,C 180,E1 -6752.506,E2 -6752.506} C_VEL
LIN {X 0,Y 481.797,Z 263.094,A -85,B 0,C 180,E1 -6755.859,E2 -6755.859} C_VEL
LIN {X 0,Y 481.751,Z 263.096,A -85,B 0,C 180,E1 -6758.387,E2 -6758.387} C_VEL
LIN {X 0,Y 481.74,Z 263.102,A -85,B 0,C 180,E1 -6761.784,E2 -6761.784} C_VEL
LIN {X 0,Y 481.731,Z 263.104,A -85,B 0,C 180,E1 -6765.223,E2 -6765.223} C_VEL
LIN {X 0,Y 481.7,Z 263.103,A -85,B 0,C 180,E1 -6768.721,E2 -6768.721} C_VEL
LIN {X 0,Y 481.634,Z 263.119,A -85,B 0,C 180,E1 -6771.394,E2 -6771.394} C_VEL
LIN {X 0,Y 481.648,Z 263.11,A -85,B 0,C 180,E1 -6774.113,E2 -6774.113} C_VEL
LIN {X 0,Y 481.734,Z 263.103,A -85,B 0,C 180,E1 -6777.138,E2 -6777.138} C_VEL
LIN {X 0,Y 481.665,Z 263.11,A -85,B 0,C 180,E1 -6779.74,E2 -6779.74} C_VEL
LIN {X 0,Y 481.659,Z 263.108,A -85,B 0,C 180,E1 -6782.673,E2 -6782.673} C_VEL
LIN {X 0,Y 481.627,Z 263.115,A -85,B 0,C 180,E1 -6785.708,E2 -6785.708} C_VEL
LIN {X 0,Y 481.657,Z 263.11,A -85,B 0,C 180,E1 -6788.858,E2 -6788.858} C_VEL
LIN {X 0,Y 481.647,Z 263.11,A -85,B 0,C 180,E1 -6791.914,E2 -6791.914} C_VEL
LIN {X 0,Y 481.645,Z 263.109,A -85,B 0,C 180,E1 -6794.457,E2 -6794.457} C_VEL
LIN {X 0,Y 481.65,Z 263.11,A -85,B 0,C 180,E1 -6797.841,E2 -6797.841} C_VEL
LIN {X 0,Y 481.656,Z 263.115,A -85,B 0,C 180,E1 -6801.141,E2 -6801.141} C_VEL
LIN {X 0,Y 481.652,Z 263.111,A -85,B 0,C 180,E1 -6804.795,E2 -6804.795} C_VEL
LIN {X 0,Y 481.658,Z 263.115,A -85,B 0,C 180,E1 -6807.326,E2 -6807.326} C_VEL
LIN {X 0,Y 481.664,Z 263.107,A -85,B 0,C 180,E1 -6810.259,E2 -6810.259} C_VEL
LIN {X 0,Y 481.73,Z 263.106,A -85,B 0,C 180,E1 -6813.112,E2 -6813.112} C_VEL
LIN {X 0,Y 481.658,Z 263.108,A -85,B 0,C 180,E1 -6815.887,E2 -6815.887} C_VEL
LIN {X 0,Y 481.687,Z 263.111,A -85,B 0,C 180,E1 -6819.028,E2 -6819.028} C_VEL
LIN {X 0,Y 481.692,Z 263.103,A -85,B 0,C 180,E1 -6822.159,E2 -6822.159} C_VEL
LIN {X 0,Y 481.728,Z 263.103,A -85,B 0,C 180,E1 -6824.776,E2 -6824.776} C_VEL
LIN {X 0,Y 481.736,Z 263.098,A -85,B 0,C 180,E1 -6828.216,E2 -6828.216} C_VEL
LIN {X 0,Y 481.747,Z 263.098,A -85,B 0,C 180,E1 -6831.612,E2 -6831.612} C_VEL
LIN {X 0,Y 481.794,Z 263.091,A -85,B 0,C 180,E1 -6834.14,E2 -6834.14} C_VEL
LIN {X 0,Y 481.913,Z 263.078,A -85,B 0,C 180,E1 -6837.493,E2 -6837.493} C_VEL
LIN {X 0,Y 481.913,Z 263.082,A -85,B 0,C 180,E1 -6840.836,E2 -6840.836} C_VEL
LIN {X 0,Y 481.914,Z 263.078,A -85,B 0,C 180,E1 -6842.508,E2 -6842.508} C_VEL
LIN {X 0,Y 481.794,Z 263.091,A -85,B 0,C 180,E1 -6845.861,E2 -6845.861} C_VEL
LIN {X 0,Y 481.75,Z 263.098,A -85,B 0,C 180,E1 -6848.389,E2 -6848.389} C_VEL
LIN {X 0,Y 481.739,Z 263.098,A -85,B 0,C 180,E1 -6851.786,E2 -6851.786} C_VEL
LIN {X 0,Y 481.731,Z 263.103,A -85,B 0,C 180,E1 -6855.225,E2 -6855.225} C_VEL
LIN {X 0,Y 481.701,Z 263.108,A -85,B 0,C 180,E1 -6858.723,E2 -6858.723} C_VEL
LIN {X 0,Y 481.634,Z 263.113,A -85,B 0,C 180,E1 -6861.396,E2 -6861.396} C_VEL
LIN {X 0,Y 481.662,Z 263.108,A -85,B 0,C 180,E1 -6864.114,E2 -6864.114} C_VEL
LIN {X 0,Y 481.736,Z 263.102,A -85,B 0,C 180,E1 -6867.14,E2 -6867.14} C_VEL
LIN {X 0,Y 481.669,Z 263.106,A -85,B 0,C 180,E1 -6869.742,E2 -6869.742} C_VEL
LIN {X 0,Y 481.662,Z 263.114,A -85,B 0,C 180,E1 -6872.675,E2 -6872.675} C_VEL
LIN {X 0,Y 481.628,Z 263.111,A -85,B 0,C 180,E1 -6875.711,E2 -6875.711} C_VEL
LIN {X 0,Y 481.661,Z 263.115,A -85,B 0,C 180,E1 -6878.86,E2 -6878.86} C_VEL
LIN {X 0,Y 481.644,Z 263.109,A -85,B 0,C 180,E1 -6881.914,E2 -6881.914} C_VEL
LIN {X 0,Y 481.647,Z 263.113,A -85,B 0,C 180,E1 -6884.459,E2 -6884.459} C_VEL
LIN {X 0,Y 481.64,Z 263.11,A -85,B 0,C 180,E1 -6887.841,E2 -6887.841} C_VEL
LIN {X 0,Y 481.674,Z 263.114,A -85,B 0,C 180,E1 -6890.653,E2 -6890.653} C_VEL
LIN {X 0,Y 481.616,Z 263.114,A -85,B 0,C 180,E1 -6893.379,E2 -6893.379} C_VEL
LIN {X 0,Y 481.705,Z 263.105,A -85,B 0,C 180,E1 -6896.331,E2 -6896.331} C_VEL
LIN {X 0,Y 481.646,Z 263.124,A -85,B 0,C 180,E1 -6898.804,E2 -6898.804} C_VEL
LIN {X 0,Y 485.585,Z 278.717,A -85,B 0,C 180,E1 -6901.239,E2 -6901.239} C_VEL
LIN {X 0,Y 486.552,Z 283.686,A -85,B 0,C 180,E1 -6901.983,E2 -6901.983} C_VEL
LIN {X 0,Y 485.503,Z 304.107,A -85,B 0,C 180,E1 -6904.722,E2 -6904.722} C_VEL
LIN {X 0,Y 484.853,Z 318.63,A -85,B 0,C 180,E1 -6906.615,E2 -6906.615} C_VEL
LIN {X 0,Y 488.73,Z 340.345,A -85,B 0,C 180,E1 -6907.186,E2 -6907.186} C_VEL
LIN {X 0,Y 486.697,Z 485.746,A -85,B 0,C 180,E1 -6909.586,E2 -6909.586} C_VEL
LIN {X 0,Y 486.244,Z 501.527,A -85,B 0,C 180,E1 -6910.015,E2 -6910.015} C_VEL
LIN {X 0,Y 485.655,Z 516.975,A -85,B 0,C 180,E1 -6910.615,E2 -6910.615} C_VEL
LIN {X 0,Y 485.041,Z 530.606,A -85,B 0,C 180,E1 -6911.303,E2 -6911.303} C_VEL
LIN {X 0,Y 484.346,Z 544.064,A -85,B 0,C 180,E1 -6912.151,E2 -6912.151} C_VEL
LIN {X 0,Y 483.678,Z 557.701,A -85,B 0,C 180,E1 -6913.207,E2 -6913.207} C_VEL
LIN {X 0,Y 483.001,Z 570.274,A -85,B 0,C 180,E1 -6914.385,E2 -6914.385} C_VEL
LIN {X 0,Y 482.408,Z 581.651,A -85,B 0,C 180,E1 -6915.662,E2 -6915.662} C_VEL
LIN {X 0,Y 481.856,Z 592.679,A -85,B 0,C 180,E1 -6917.15,E2 -6917.15} C_VEL
LIN {X 0,Y 481.521,Z 601.857,A -85,B 0,C 180,E1 -6918.637,E2 -6918.637} C_VEL
LIN {X 0,Y 481.244,Z 608.434,A -85,B 0,C 180,E1 -6919.908,E2 -6919.908} C_VEL
LIN {X 0,Y 481.039,Z 615.706,A -85,B 0,C 180,E1 -6921.6,E2 -6921.6} C_VEL
LIN {X 0,Y 480.953,Z 621.421,A -85,B 0,C 180,E1 -6923.288,E2 -6923.288} C_VEL
LIN {X 0,Y 480.859,Z 625.731,A -85,B 0,C 180,E1 -6924.97,E2 -6924.97} C_VEL
LIN {X 0,Y 480.88,Z 628.749,A -85,B 0,C 180,E1 -6926.65,E2 -6926.65} C_VEL
LIN {X 0,Y 480.822,Z 630.532,A -85,B 0,C 180,E1 -6928.326,E2 -6928.326} C_VEL
LIN {X 0,Y 480.743,Z 631.108,A -85,B 0,C 180,E1 -6930.001,E2 -6930.001} C_VEL
LIN {X 0,Y 480.823,Z 630.449,A -85,B 0,C 180,E1 -6931.676,E2 -6931.676} C_VEL
LIN {X 0,Y 480.881,Z 628.586,A -85,B 0,C 180,E1 -6933.352,E2 -6933.352} C_VEL
LIN {X 0,Y 480.869,Z 625.481,A -85,B 0,C 180,E1 -6935.032,E2 -6935.032} C_VEL
LIN {X 0,Y 480.91,Z 621.061,A -85,B 0,C 180,E1 -6936.715,E2 -6936.715} C_VEL
LIN {X 0,Y 481.041,Z 615.205,A -85,B 0,C 180,E1 -6938.402,E2 -6938.402} C_VEL
LIN {X 0,Y 481.234,Z 607.754,A -85,B 0,C 180,E1 -6940.094,E2 -6940.094} C_VEL
LIN {X 0,Y 481.524,Z 599.756,A -85,B 0,C 180,E1 -6941.578,E2 -6941.578} C_VEL
LIN {X 0,Y 481.904,Z 590.098,A -85,B 0,C 180,E1 -6943.066,E2 -6943.066} C_VEL
LIN {X 0,Y 482.301,Z 580.26,A -85,B 0,C 180,E1 -6944.344,E2 -6944.344} C_VEL
LIN {X 0,Y 482.862,Z 568.558,A -85,B 0,C 180,E1 -6945.622,E2 -6945.622} C_VEL
LIN {X 0,Y 483.509,Z 555.667,A -85,B 0,C 180,E1 -6946.793,E2 -6946.793} C_VEL
LIN {X 0,Y 484.122,Z 543.035,A -85,B 0,C 180,E1 -6947.751,E2 -6947.751} C_VEL
LIN {X 0,Y 484.746,Z 529.384,A -85,B 0,C 180,E1 -6948.601,E2 -6948.601} C_VEL
LIN {X 0,Y 485.409,Z 514.472,A -85,B 0,C 180,E1 -6949.342,E2 -6949.342} C_VEL
LIN {X 0,Y 485.995,Z 498.388,A -85,B 0,C 180,E1 -6949.946,E2 -6949.946} C_VEL
LIN {X 0,Y 486.436,Z 483.169,A -85,B 0,C 180,E1 -6950.345,E2 -6950.345} C_VEL
LIN {X 0,Y 488.193,Z 370.417,A -85,B 0,C 180,E1 -6952.287,E2 -6952.287} C_VEL
LIN {X 0,Y 488.712,Z 339.874,A -85,B 0,C 180,E1 -6952.848,E2 -6952.848} C_VEL
LIN {X 0,Y 484.981,Z 317.317,A -85,B 0,C 180,E1 -6953.507,E2 -6953.507} C_VEL
LIN {X 0,Y 484.573,Z 314.94,A -85,B 0,C 180,E1 -6953.594,E2 -6953.594} C_VEL
LIN {X 0,Y 485.878,Z 290.835,A -85,B 0,C 180,E1 -6956.874,E2 -6956.874} C_VEL
LIN {X 0,Y 486.24,Z 281.808,A -85,B 0,C 180,E1 -6958.154,E2 -6958.154} C_VEL
LIN {X 0,Y 484.016,Z 271.691,A -85,B 0,C 180,E1 -6959.824,E2 -6959.824} C_VEL
LIN {X 0,Y 481.66,Z 263.117,A -85,B 0,C 180,E1 -6961.381,E2 -6961.381} C_VEL
LIN {X 0,Y 481.703,Z 263.111,A -85,B 0,C 180,E1 -6963.734,E2 -6963.734} C_VEL
LIN {X 0,Y 481.631,Z 263.119,A -85,B 0,C 180,E1 -6966.747,E2 -6966.747} C_VEL
LIN {X 0,Y 481.683,Z 263.109,A -85,B 0,C 180,E1 -6969.941,E2 -6969.941} C_VEL
LIN {X 0,Y 481.645,Z 263.116,A -85,B 0,C 180,E1 -6973.3,E2 -6973.3} C_VEL
LIN {X 0,Y 481.664,Z 263.111,A -85,B 0,C 180,E1 -6975.641,E2 -6975.641} C_VEL
LIN {X 0,Y 481.662,Z 263.115,A -85,B 0,C 180,E1 -6978.958,E2 -6978.958} C_VEL
LIN {X 0,Y 481.656,Z 263.113,A -85,B 0,C 180,E1 -6981.994,E2 -6981.994} C_VEL
LIN {X 0,Y 481.694,Z 263.108,A -85,B 0,C 180,E1 -6985.318,E2 -6985.318} C_VEL
LIN {X 0,Y 481.651,Z 263.117,A -85,B 0,C 180,E1 -6988.312,E2 -6988.312} C_VEL
LIN {X 0,Y 481.68,Z 263.111,A -85,B 0,C 180,E1 -6991.217,E2 -6991.217} C_VEL
LIN {X 0,Y 481.682,Z 263.112,A -85,B 0,C 180,E1 -6994.041,E2 -6994.041} C_VEL
LIN {X 0,Y 481.711,Z 263.234,A -85,B 0,C 180,E1 -6994.707,E2 -6994.707} C_VEL
LIN {X 0,Y 483.651,Z 271.127,A -85,B 0,C 180,E1 -6996.463,E2 -6996.463} C_VEL
LIN {X 0,Y 489.12,Z 283.755,A -85,B 0,C 180,E1 -6997.058,E2 -6997.058} C_VEL
LIN {X 0,Y 489.429,Z 286.521,A -85,B 0,C 180,E1 -6997.132,E2 -6997.132} C_VEL
LIN {X 0,Y 487.319,Z 388.91,A -85,B 0,C 180,E1 -6998.977,E2 -6998.977} C_VEL
LIN {X 0,Y 486.657,Z 435.089,A -85,B 0,C 180,E1 -6999.786,E2 -6999.786} C_VEL
LIN {X 0,Y 486.285,Z 450.548,A -85,B 0,C 180,E1 -7000.224,E2 -7000.224} C_VEL
LIN {X 0,Y 485.819,Z 465.842,A -85,B 0,C 180,E1 -7000.84,E2 -7000.84} C_VEL
LIN {X 0,Y 485.332,Z 479.128,A -85,B 0,C 180,E1 -7001.532,E2 -7001.532} C_VEL
LIN {X 0,Y 484.771,Z 492.315,A -85,B 0,C 180,E1 -7002.383,E2 -7002.383} C_VEL
LIN {X 0,Y 484.083,Z 505.007,A -85,B 0,C 180,E1 -7003.377,E2 -7003.377} C_VEL
LIN {X 0,Y 483.434,Z 517.922,A -85,B 0,C 180,E1 -7004.614,E2 -7004.614} C_VEL
LIN {X 0,Y 482.89,Z 528.995,A -85,B 0,C 180,E1 -7005.89,E2 -7005.89} C_VEL
LIN {X 0,Y 482.328,Z 538.338,A -85,B 0,C 180,E1 -7007.161,E2 -7007.161} C_VEL
LIN {X 0,Y 481.96,Z 547.423,A -85,B 0,C 180,E1 -7008.646,E2 -7008.646} C_VEL
LIN {X 0,Y 481.586,Z 553.916,A -85,B 0,C 180,E1 -7009.914,E2 -7009.914} C_VEL
LIN {X 0,Y 481.306,Z 561.092,A -85,B 0,C 180,E1 -7011.603,E2 -7011.603} C_VEL
LIN {X 0,Y 481.111,Z 566.997,A -85,B 0,C 180,E1 -7013.385,E2 -7013.385} C_VEL
LIN {X 0,Y 480.902,Z 570.944,A -85,B 0,C 180,E1 -7014.969,E2 -7014.969} C_VEL
LIN {X 0,Y 480.949,Z 573.892,A -85,B 0,C 180,E1 -7016.648,E2 -7016.648} C_VEL
LIN {X 0,Y 480.825,Z 575.658,A -85,B 0,C 180,E1 -7018.324,E2 -7018.324} C_VEL
LIN {X 0,Y 480.748,Z 576.242,A -85,B 0,C 180,E1 -7019.999,E2 -7019.999} C_VEL
LIN {X 0,Y 480.825,Z 575.622,A -85,B 0,C 180,E1 -7021.674,E2 -7021.674} C_VEL
LIN {X 0,Y 480.939,Z 573.848,A -85,B 0,C 180,E1 -7023.35,E2 -7023.35} C_VEL
LIN {X 0,Y 480.893,Z 570.892,A -85,B 0,C 180,E1 -7025.03,E2 -7025.03} C_VEL
LIN {X 0,Y 481.093,Z 567.003,A -85,B 0,C 180,E1 -7026.596,E2 -7026.596} C_VEL
LIN {X 0,Y 481.254,Z 561.069,A -85,B 0,C 180,E1 -7028.396,E2 -7028.396} C_VEL
LIN {X 0,Y 481.524,Z 553.943,A -85,B 0,C 180,E1 -7030.086,E2 -7030.086} C_VEL
LIN {X 0,Y 481.914,Z 546.286,A -85,B 0,C 180,E1 -7031.567,E2 -7031.567} C_VEL
LIN {X 0,Y 482.359,Z 537.041,A -85,B 0,C 180,E1 -7033.051,E2 -7033.051} C_VEL
LIN {X 0,Y 482.86,Z 527.605,A -85,B 0,C 180,E1 -7034.325,E2 -7034.325} C_VEL
LIN {X 0,Y 483.477,Z 515.349,A -85,B 0,C 180,E1 -7035.707,E2 -7035.707} C_VEL
LIN {X 0,Y 484.189,Z 502.807,A -85,B 0,C 180,E1 -7036.875,E2 -7036.875} C_VEL
LIN {X 0,Y 484.79,Z 490.489,A -85,B 0,C 180,E1 -7037.832,E2 -7037.832} C_VEL
LIN {X 0,Y 485.423,Z 477.147,A -85,B 0,C 180,E1 -7038.682,E2 -7038.682} C_VEL
LIN {X 0,Y 486.026,Z 462.514,A -85,B 0,C 180,E1 -7039.425,E2 -7039.425} C_VEL
LIN {X 0,Y 486.503,Z 447.292,A -85,B 0,C 180,E1 -7040.012,E2 -7040.012} C_VEL
LIN {X 0,Y 486.888,Z 431.61,A -85,B 0,C 180,E1 -7040.434,E2 -7040.434} C_VEL
LIN {X 0,Y 488.857,Z 284.463,A -85,B 0,C 180,E1 -7042.873,E2 -7042.873} C_VEL
LIN {X 0,Y 487.318,Z 279.262,A -85,B 0,C 180,E1 -7043.04,E2 -7043.04} C_VEL
LIN {X 0,Y 482.504,Z 266.924,A -85,B 0,C 180,E1 -7043.51,E2 -7043.51} C_VEL
LIN {X 0,Y 481.674,Z 263.114,A -85,B 0,C 180,E1 -7044.255,E2 -7044.255} C_VEL
LIN {X 0,Y 481.695,Z 263.105,A -85,B 0,C 180,E1 -7047.126,E2 -7047.126} C_VEL
LIN {X 0,Y 481.673,Z 263.113,A -85,B 0,C 180,E1 -7049.74,E2 -7049.74} C_VEL
LIN {X 0,Y 481.672,Z 263.106,A -85,B 0,C 180,E1 -7052.673,E2 -7052.673} C_VEL
LIN {X 0,Y 481.66,Z 263.108,A -85,B 0,C 180,E1 -7055.203,E2 -7055.203} C_VEL
LIN {X 0,Y 481.668,Z 263.106,A -85,B 0,C 180,E1 -7058.858,E2 -7058.858} C_VEL
LIN {X 0,Y 481.645,Z 263.117,A -85,B 0,C 180,E1 -7061.911,E2 -7061.911} C_VEL
LIN {X 0,Y 481.651,Z 263.11,A -85,B 0,C 180,E1 -7064.385,E2 -7064.385} C_VEL
LIN {X 0,Y 480.994,Z 263.192,A -85,B 0,C 180,E1 -7065.083,E2 -7065.083} C_VEL
LIN {X 0,Y 478.142,Z 263.55,A -85,B 0,C 180,E1 -7066.216,E2 -7066.216} C_VEL
LIN {X 0,Y 475.727,Z 263.854,A -85,B 0,C 180,E1 -7067.13,E2 -7067.13} C_VEL
LIN {X 0,Y 474.696,Z 263.983,A -85,B 0,C 180,E1 -7067.836,E2 -7067.836} C_VEL
LIN {X 0,Y 474.616,Z 263.989,A -85,B 0,C 180,E1 -7068.075,E2 -7068.075} C_VEL
LIN {X 0,Y 474.63,Z 263.984,A -85,B 0,C 180,E1 -7070.452,E2 -7070.452} C_VEL
LIN {X 0,Y 474.585,Z 263.996,A -85,B 0,C 180,E1 -7073.675,E2 -7073.675} C_VEL
LIN {X 0,Y 474.621,Z 263.984,A -85,B 0,C 180,E1 -7076.777,E2 -7076.777} C_VEL
LIN {X 0,Y 474.599,Z 263.995,A -85,B 0,C 180,E1 -7079.768,E2 -7079.768} C_VEL
LIN {X 0,Y 474.632,Z 263.983,A -85,B 0,C 180,E1 -7082.675,E2 -7082.675} C_VEL
LIN {X 0,Y 474.632,Z 263.989,A -85,B 0,C 180,E1 -7085.505,E2 -7085.505} C_VEL
LIN {X 0,Y 474.665,Z 263.981,A -85,B 0,C 180,E1 -7089.184,E2 -7089.184} C_VEL
LIN {X 0,Y 474.64,Z 263.987,A -85,B 0,C 180,E1 -7091.883,E2 -7091.883} C_VEL
LIN {X 0,Y 474.693,Z 263.975,A -85,B 0,C 180,E1 -7094.543,E2 -7094.543} C_VEL
LIN {X 0,Y 474.697,Z 263.978,A -85,B 0,C 180,E1 -7098.036,E2 -7098.036} C_VEL
LIN {X 0,Y 474.721,Z 263.979,A -85,B 0,C 180,E1 -7101.485,E2 -7101.485} C_VEL
LIN {X 0,Y 474.761,Z 263.969,A -85,B 0,C 180,E1 -7104.051,E2 -7104.051} C_VEL
LIN {X 0,Y 474.884,Z 263.958,A -85,B 0,C 180,E1 -7107.454,E2 -7107.454} C_VEL
LIN {X 0,Y 474.848,Z 263.957,A -85,B 0,C 180,E1 -7110.847,E2 -7110.847} C_VEL
LIN {X 0,Y 474.883,Z 263.952,A -85,B 0,C 180,E1 -7112.543,E2 -7112.543} C_VEL
LIN {X 0,Y 474.76,Z 263.97,A -85,B 0,C 180,E1 -7115.947,E2 -7115.947} C_VEL
LIN {X 0,Y 474.716,Z 263.972,A -85,B 0,C 180,E1 -7118.512,E2 -7118.512} C_VEL
LIN {X 0,Y 474.693,Z 263.978,A -85,B 0,C 180,E1 -7121.961,E2 -7121.961} C_VEL
LIN {X 0,Y 474.688,Z 263.985,A -85,B 0,C 180,E1 -7125.455,E2 -7125.455} C_VEL
LIN {X 0,Y 474.653,Z 263.983,A -85,B 0,C 180,E1 -7129.009,E2 -7129.009} C_VEL
LIN {X 0,Y 474.576,Z 263.994,A -85,B 0,C 180,E1 -7131.728,E2 -7131.728} C_VEL
LIN {X 0,Y 474.628,Z 263.983,A -85,B 0,C 180,E1 -7134.493,E2 -7134.493} C_VEL
LIN {X 0,Y 474.686,Z 263.984,A -85,B 0,C 180,E1 -7137.338,E2 -7137.338} C_VEL
LIN {X 0,Y 474.591,Z 263.99,A -85,B 0,C 180,E1 -7140.81,E2 -7140.81} C_VEL
LIN {X 0,Y 474.624,Z 263.985,A -85,B 0,C 180,E1 -7143.983,E2 -7143.983} C_VEL
LIN {X 0,Y 474.56,Z 263.995,A -85,B 0,C 180,E1 -7146.899,E2 -7146.899} C_VEL
LIN {X 0,Y 474.613,Z 263.989,A -85,B 0,C 180,E1 -7149.647,E2 -7149.647} C_VEL
LIN {X 0,Y 474.62,Z 263.988,A -85,B 0,C 180,E1 -7152.931,E2 -7152.931} C_VEL
LIN {X 0,Y 474.601,Z 263.988,A -85,B 0,C 180,E1 -7155.896,E2 -7155.896} C_VEL
LIN {X 0,Y 474.617,Z 263.99,A -85,B 0,C 180,E1 -7159.04,E2 -7159.04} C_VEL
LIN {X 0,Y 474.595,Z 263.99,A -85,B 0,C 180,E1 -7161.704,E2 -7161.704} C_VEL
LIN {X 0,Y 474.614,Z 263.987,A -85,B 0,C 180,E1 -7164.726,E2 -7164.726} C_VEL
LIN {X 0,Y 474.622,Z 263.986,A -85,B 0,C 180,E1 -7167.788,E2 -7167.788} C_VEL
LIN {X 0,Y 474.609,Z 263.99,A -85,B 0,C 180,E1 -7170.884,E2 -7170.884} C_VEL
LIN {X 0,Y 474.645,Z 263.984,A -85,B 0,C 180,E1 -7173.628,E2 -7173.628} C_VEL
LIN {X 0,Y 474.62,Z 263.986,A -85,B 0,C 180,E1 -7176.642,E2 -7176.642} C_VEL
LIN {X 0,Y 474.642,Z 263.982,A -85,B 0,C 180,E1 -7180.09,E2 -7180.09} C_VEL
LIN {X 0,Y 474.635,Z 263.986,A -85,B 0,C 180,E1 -7182.775,E2 -7182.775} C_VEL
LIN {X 0,Y 474.633,Z 263.987,A -85,B 0,C 180,E1 -7185.421,E2 -7185.421} C_VEL
LIN {X 0,Y 474.689,Z 263.976,A -85,B 0,C 180,E1 -7188.038,E2 -7188.038} C_VEL
LIN {X 0,Y 474.713,Z 263.976,A -85,B 0,C 180,E1 -7191.487,E2 -7191.487} C_VEL
LIN {X 0,Y 474.756,Z 263.967,A -85,B 0,C 180,E1 -7194.053,E2 -7194.053} C_VEL
LIN {X 0,Y 474.879,Z 263.955,A -85,B 0,C 180,E1 -7197.456,E2 -7197.456} C_VEL
LIN {X 0,Y 474.864,Z 263.96,A -85,B 0,C 180,E1 -7200.849,E2 -7200.849} C_VEL
LIN {X 0,Y 474.88,Z 263.955,A -85,B 0,C 180,E1 -7202.545,E2 -7202.545} C_VEL
LIN {X 0,Y 474.757,Z 263.967,A -85,B 0,C 180,E1 -7205.948,E2 -7205.948} C_VEL
LIN {X 0,Y 474.716,Z 263.975,A -85,B 0,C 180,E1 -7208.514,E2 -7208.514} C_VEL
LIN {X 0,Y 474.692,Z 263.975,A -85,B 0,C 180,E1 -7211.963,E2 -7211.963} C_VEL
LIN {X 0,Y 474.688,Z 263.978,A -85,B 0,C 180,E1 -7215.457,E2 -7215.457} C_VEL
LIN {X 0,Y 474.654,Z 263.987,A -85,B 0,C 180,E1 -7219.011,E2 -7219.011} C_VEL
LIN {X 0,Y 474.577,Z 263.99,A -85,B 0,C 180,E1 -7221.73,E2 -7221.73} C_VEL
LIN {X 0,Y 474.644,Z 263.985,A -85,B 0,C 180,E1 -7224.494,E2 -7224.494} C_VEL
LIN {X 0,Y 474.671,Z 263.98,A -85,B 0,C 180,E1 -7227.335,E2 -7227.335} C_VEL
LIN {X 0,Y 474.595,Z 263.989,A -85,B 0,C 180,E1 -7230.231,E2 -7230.231} C_VEL
LIN {X 0,Y 474.633,Z 263.986,A -85,B 0,C 180,E1 -7233.221,E2 -7233.221} C_VEL
LIN {X 0,Y 474.58,Z 263.992,A -85,B 0,C 180,E1 -7236.325,E2 -7236.325} C_VEL
LIN {X 0,Y 474.609,Z 263.986,A -85,B 0,C 180,E1 -7239.647,E2 -7239.647} C_VEL
LIN {X 0,Y 474.606,Z 263.992,A -85,B 0,C 180,E1 -7242.936,E2 -7242.936} C_VEL
LIN {X 0,Y 474.599,Z 263.987,A -85,B 0,C 180,E1 -7245.896,E2 -7245.896} C_VEL
LIN {X 0,Y 474.621,Z 263.99,A -85,B 0,C 180,E1 -7249.042,E2 -7249.042} C_VEL
LIN {X 0,Y 474.601,Z 263.988,A -85,B 0,C 180,E1 -7251.706,E2 -7251.706} C_VEL
LIN {X 0,Y 474.616,Z 263.989,A -85,B 0,C 180,E1 -7254.727,E2 -7254.727} C_VEL
LIN {X 0,Y 474.63,Z 263.985,A -85,B 0,C 180,E1 -7257.789,E2 -7257.789} C_VEL
LIN {X 0,Y 474.626,Z 264.114,A -85,B 0,C 180,E1 -7258.507,E2 -7258.507} C_VEL
LIN {X 0,Y 478.936,Z 281.181,A -85,B 0,C 180,E1 -7261.209,E2 -7261.209} C_VEL
LIN {X 0,Y 479.704,Z 284.843,A -85,B 0,C 180,E1 -7261.767,E2 -7261.767} C_VEL
LIN {X 0,Y 478.907,Z 300.314,A -85,B 0,C 180,E1 -7263.882,E2 -7263.882} C_VEL
LIN {X 0,Y 477.994,Z 317.983,A -85,B 0,C 180,E1 -7266.259,E2 -7266.259} C_VEL
LIN {X 0,Y 482.169,Z 341.6,A -85,B 0,C 180,E1 -7266.894,E2 -7266.894} C_VEL
LIN {X 0,Y 479.955,Z 485.161,A -85,B 0,C 180,E1 -7269.314,E2 -7269.314} C_VEL
LIN {X 0,Y 479.453,Z 501.211,A -85,B 0,C 180,E1 -7269.757,E2 -7269.757} C_VEL
LIN {X 0,Y 478.869,Z 515.887,A -85,B 0,C 180,E1 -7270.329,E2 -7270.329} C_VEL
LIN {X 0,Y 478.207,Z 529.629,A -85,B 0,C 180,E1 -7271.026,E2 -7271.026} C_VEL
LIN {X 0,Y 477.526,Z 543.183,A -85,B 0,C 180,E1 -7271.887,E2 -7271.887} C_VEL
LIN {X 0,Y 476.784,Z 555.713,A -85,B 0,C 180,E1 -7272.855,E2 -7272.855} C_VEL
LIN {X 0,Y 476.152,Z 568.5,A -85,B 0,C 180,E1 -7274.045,E2 -7274.045} C_VEL
LIN {X 0,Y 475.485,Z 579.198,A -85,B 0,C 180,E1 -7275.23,E2 -7275.23} C_VEL
LIN {X 0,Y 475.027,Z 589.12,A -85,B 0,C 180,E1 -7276.526,E2 -7276.526} C_VEL
LIN {X 0,Y 474.469,Z 598.829,A -85,B 0,C 180,E1 -7278.033,E2 -7278.033} C_VEL
LIN {X 0,Y 474.284,Z 606.914,A -85,B 0,C 180,E1 -7279.543,E2 -7279.543} C_VEL
LIN {X 0,Y 474.005,Z 613.594,A -85,B 0,C 180,E1 -7281.045,E2 -7281.045} C_VEL
LIN {X 0,Y 473.895,Z 619.712,A -85,B 0,C 180,E1 -7282.759,E2 -7282.759} C_VEL
LIN {X 0,Y 473.809,Z 623.32,A -85,B 0,C 180,E1 -7284.041,E2 -7284.041} C_VEL
LIN {X 0,Y 473.735,Z 626.986,A -85,B 0,C 180,E1 -7285.747,E2 -7285.747} C_VEL
LIN {X 0,Y 473.778,Z 629.391,A -85,B 0,C 180,E1 -7287.451,E2 -7287.451} C_VEL
LIN {X 0,Y 473.687,Z 630.572,A -85,B 0,C 180,E1 -7289.151,E2 -7289.151} C_VEL
LIN {X 0,Y 473.687,Z 630.522,A -85,B 0,C 180,E1 -7290.851,E2 -7290.851} C_VEL
LIN {X 0,Y 473.802,Z 629.249,A -85,B 0,C 180,E1 -7292.552,E2 -7292.552} C_VEL
LIN {X 0,Y 473.742,Z 626.745,A -85,B 0,C 180,E1 -7294.255,E2 -7294.255} C_VEL
LIN {X 0,Y 473.816,Z 622.972,A -85,B 0,C 180,E1 -7295.961,E2 -7295.961} C_VEL
LIN {X 0,Y 473.91,Z 617.819,A -85,B 0,C 180,E1 -7297.671,E2 -7297.671} C_VEL
LIN {X 0,Y 474.026,Z 611.137,A -85,B 0,C 180,E1 -7299.387,E2 -7299.387} C_VEL
LIN {X 0,Y 474.339,Z 603.931,A -85,B 0,C 180,E1 -7300.89,E2 -7300.89} C_VEL
LIN {X 0,Y 474.625,Z 595.15,A -85,B 0,C 180,E1 -7302.41,E2 -7302.41} C_VEL
LIN {X 0,Y 475.103,Z 584.688,A -85,B 0,C 180,E1 -7303.91,E2 -7303.91} C_VEL
LIN {X 0,Y 475.645,Z 573.927,A -85,B 0,C 180,E1 -7305.206,E2 -7305.206} C_VEL
LIN {X 0,Y 476.262,Z 561.856,A -85,B 0,C 180,E1 -7306.427,E2 -7306.427} C_VEL
LIN {X 0,Y 476.914,Z 548.038,A -85,B 0,C 180,E1 -7307.585,E2 -7307.585} C_VEL
LIN {X 0,Y 477.673,Z 533.869,A -85,B 0,C 180,E1 -7308.553,E2 -7308.553} C_VEL
LIN {X 0,Y 478.392,Z 519.18,A -85,B 0,C 180,E1 -7309.359,E2 -7309.359} C_VEL
LIN {X 0,Y 479.019,Z 504.006,A -85,B 0,C 180,E1 -7310.003,E2 -7310.003} C_VEL
LIN {X 0,Y 479.57,Z 488.483,A -85,B 0,C 180,E1 -7310.484,E2 -7310.484} C_VEL
LIN {X 0,Y 479.93,Z 469.858,A -85,B 0,C 180,E1 -7310.857,E2 -7310.857} C_VEL
LIN {X 0,Y 481.595,Z 377.793,A -85,B 0,C 180,E1 -7312.481,E2 -7312.481} C_VEL
LIN {X 0,Y 482.24,Z 340.766,A -85,B 0,C 180,E1 -7313.185,E2 -7313.185} C_VEL
LIN {X 0,Y 478.649,Z 318.82,A -85,B 0,C 180,E1 -7313.853,E2 -7313.853} C_VEL
LIN {X 0,Y 477.842,Z 314.359,A -85,B 0,C 180,E1 -7314.005,E2 -7314.005} C_VEL
LIN {X 0,Y 479.244,Z 290.894,A -85,B 0,C 180,E1 -7317.277,E2 -7317.277} C_VEL
LIN {X 0,Y 479.594,Z 284.485,A -85,B 0,C 180,E1 -7318.203,E2 -7318.203} C_VEL
LIN {X 0,Y 477.687,Z 275.155,A -85,B 0,C 180,E1 -7319.768,E2 -7319.768} C_VEL
LIN {X 0,Y 474.605,Z 263.994,A -85,B 0,C 180,E1 -7321.84,E2 -7321.84} C_VEL
LIN {X 0,Y 474.637,Z 263.99,A -85,B 0,C 180,E1 -7324.242,E2 -7324.242} C_VEL
LIN {X 0,Y 474.595,Z 263.995,A -85,B 0,C 180,E1 -7327.384,E2 -7327.384} C_VEL
LIN {X 0,Y 474.633,Z 263.988,A -85,B 0,C 180,E1 -7329.648,E2 -7329.648} C_VEL
LIN {X 0,Y 474.621,Z 263.992,A -85,B 0,C 180,E1 -7332.935,E2 -7332.935} C_VEL
LIN {X 0,Y 474.615,Z 263.989,A -85,B 0,C 180,E1 -7335.895,E2 -7335.895} C_VEL
LIN {X 0,Y 474.634,Z 263.989,A -85,B 0,C 180,E1 -7339.041,E2 -7339.041} C_VEL
LIN {X 0,Y 474.613,Z 263.989,A -85,B 0,C 180,E1 -7341.705,E2 -7341.705} C_VEL
LIN {X 0,Y 474.628,Z 263.991,A -85,B 0,C 180,E1 -7344.726,E2 -7344.726} C_VEL
LIN {X 0,Y 474.642,Z 263.987,A -85,B 0,C 180,E1 -7347.788,E2 -7347.788} C_VEL
LIN {X 0,Y 474.613,Z 263.993,A -85,B 0,C 180,E1 -7350.888,E2 -7350.888} C_VEL
LIN {X 0,Y 474.664,Z 263.986,A -85,B 0,C 180,E1 -7354.166,E2 -7354.166} C_VEL
LIN {X 0,Y 476.699,Z 272.053,A -85,B 0,C 180,E1 -7356.026,E2 -7356.026} C_VEL
LIN {X 0,Y 483.026,Z 286.221,A -85,B 0,C 180,E1 -7356.743,E2 -7356.743} C_VEL
LIN {X 0,Y 480.807,Z 385.015,A -85,B 0,C 180,E1 -7358.594,E2 -7358.594} C_VEL
LIN {X 0,Y 479.991,Z 435.4,A -85,B 0,C 180,E1 -7359.501,E2 -7359.501} C_VEL
LIN {X 0,Y 479.601,Z 450.963,A -85,B 0,C 180,E1 -7359.95,E2 -7359.95} C_VEL
LIN {X 0,Y 479.104,Z 465.951,A -85,B 0,C 180,E1 -7360.56,E2 -7360.56} C_VEL
LIN {X 0,Y 478.588,Z 479.281,A -85,B 0,C 180,E1 -7361.262,E2 -7361.262} C_VEL
LIN {X 0,Y 478.003,Z 492.515,A -85,B 0,C 180,E1 -7362.126,E2 -7362.126} C_VEL
LIN {X 0,Y 477.236,Z 505.783,A -85,B 0,C 180,E1 -7363.182,E2 -7363.182} C_VEL
LIN {X 0,Y 476.555,Z 518.185,A -85,B 0,C 180,E1 -7364.386,E2 -7364.386} C_VEL
LIN {X 0,Y 475.984,Z 529.295,A -85,B 0,C 180,E1 -7365.681,E2 -7365.681} C_VEL
LIN {X 0,Y 475.378,Z 538.651,A -85,B 0,C 180,E1 -7366.97,E2 -7366.97} C_VEL
LIN {X 0,Y 474.982,Z 547.755,A -85,B 0,C 180,E1 -7368.477,E2 -7368.477} C_VEL
LIN {X 0,Y 474.577,Z 554.278,A -85,B 0,C 180,E1 -7369.763,E2 -7369.763} C_VEL
LIN {X 0,Y 474.285,Z 561.471,A -85,B 0,C 180,E1 -7371.478,E2 -7371.478} C_VEL
LIN {X 0,Y 474.067,Z 567.105,A -85,B 0,C 180,E1 -7373.188,E2 -7373.188} C_VEL
LIN {X 0,Y 474.032,Z 569.387,A -85,B 0,C 180,E1 -7374.042,E2 -7374.042} C_VEL
LIN {X 0,Y 473.91,Z 572.976,A -85,B 0,C 180,E1 -7375.747,E2 -7375.747} C_VEL
LIN {X 0,Y 473.876,Z 575.331,A -85,B 0,C 180,E1 -7377.449,E2 -7377.449} C_VEL
LIN {X 0,Y 473.691,Z 576.515,A -85,B 0,C 180,E1 -7379.149,E2 -7379.149} C_VEL
LIN {X 0,Y 473.691,Z 576.478,A -85,B 0,C 180,E1 -7380.849,E2 -7380.849} C_VEL
LIN {X 0,Y 473.874,Z 575.264,A -85,B 0,C 180,E1 -7382.549,E2 -7382.549} C_VEL
LIN {X 0,Y 473.89,Z 572.886,A -85,B 0,C 180,E1 -7384.252,E2 -7384.252} C_VEL
LIN {X 0,Y 474.02,Z 569.272,A -85,B 0,C 180,E1 -7385.956,E2 -7385.956} C_VEL
LIN {X 0,Y 474.103,Z 564.346,A -85,B 0,C 180,E1 -7387.666,E2 -7387.666} C_VEL
LIN {X 0,Y 474.343,Z 557.969,A -85,B 0,C 180,E1 -7389.379,E2 -7389.379} C_VEL
LIN {X 0,Y 474.779,Z 549.939,A -85,B 0,C 180,E1 -7391.094,E2 -7391.094} C_VEL
